(* IEC 61131-3 sources: F100R_S278_Temperville/MyController.device.xml.v3^/Plc Logic.plclogic.xml.v3^/Application.application.xml.v3^/04_PID, 11 files *)

(* ---- A_PincipalRampa.prg.st ---- *)
PROGRAM A_PincipalRampa

IF NOT xTesteResistencias AND NOT xTesteEntradaSaidas THEN
	B_RampaPatamar();
	C_AquecimentoReceita();
ELSE
	E_Termperaturas();
END_IF

(* ---- A_PrincipalPid.prg.st ---- *)
PROGRAM A_PrincipalPid
VAR

END_VAR

IF NOT xTesteResistencias AND NOT xTesteEntradaSaidas THEN
	D_CtrlResistInferiores();
	D_CtrlResistSuperiores();
	//SR_Main();
ELSE
	E_Termperaturas();
END_IF

D_CtrlResist();
C_StandByTemperaturas();
A_TemperaturaGeral();
D_ConvecVentEnt();
D_ConvecVentSai();

(* ---- A_TemperaturaGeral.prg.st ---- *)
PROGRAM A_TemperaturaGeral
VAR
	IndexGTI: INT;
	IndexGPI: INT;
	IndexGTS: INT;
	IndexGPS: INT;
	IndexGTIS: INT;
	IndexGPIS: INT;
	IndexGTSS: INT;
	IndexGPSS: INT;
END_VAR

// ATUALIZAÇÃO DAS TEMPERATURAS E PERCENTAGENS PELA TEMPERATURA GERAL

IF NOT xBloqueioCargaEnvioRec THEN
	// Temperaturas Inferiores
	IF rSetTemperaturaInferiorGeral <> rSetTemperaturaInferiorGeralAux THEN
		FOR IndexGTI:=1 TO iNumResistencias DO
			rSetTemperaturaInferior[IndexGTI]:=rSetTemperaturaInferiorGeral;
		END_FOR
		rSetTemperaturaInferiorGeralAux:=rSetTemperaturaInferiorGeral;
	END_IF

	//Percentagens Inferiores
	IF rSetPorcentagemInferiorGeral <> rSetPorcentagemInferiorGeralAux THEN
		FOR IndexGPI:=1 TO iNumResistencias DO
			rSetPorcentagemInferior[IndexGPI]:=rSetPorcentagemInferiorGeral;
		END_FOR
		rSetPorcentagemInferiorGeralAux:=rSetPorcentagemInferiorGeral;
	END_IF

	//Temperaturas Superiores
	IF rSetTemperaturaSuperiorGeral <> rSetTemperaturaSuperiorGeralAux THEN
		FOR IndexGTS:=1 TO iNumResistencias DO
			rSetTemperaturaSuperior[IndexGTS]:=rSetTemperaturaSuperiorGeral;
		END_FOR
		rSetTemperaturaSuperiorGeralAux:=rSetTemperaturaSuperiorGeral;
	END_IF

	//Percentagens Superiores
	IF rSetPorcentagemSuperiorGeral <> rSetPorcentagemSuperiorGeralAux THEN
		FOR IndexGPS:=1 TO iNumResistencias DO
			rSetPorcentagemSuperior[IndexGPS]:=rSetPorcentagemSuperiorGeral;
		END_FOR
		rSetPorcentagemSuperiorGeralAux:=rSetPorcentagemSuperiorGeral;
	END_IF
END_IF

// INCREMENTA/DECREMENTA MESMO VALOR EM TODAS AS TEMPERATURAS

// Temperaturas Inferiores
	IF xBtHabIncremento THEN
		FOR IndexGTIS:=1 TO iNumResistencias DO
			rSetTemperaturaInferior[IndexGTIS]:=rSetTemperaturaInferior[IndexGTIS]+rIncrementoTemperInf;
			rSetPorcentagemInferior[IndexGTIS]:=rSetPorcentagemInferior[IndexGTIS]+rIncrementoPotenciaInf;
			rSetTemperaturaSuperior[IndexGTIS]:=rSetTemperaturaSuperior[IndexGTIS]+rIncrementoTemperSup;
			rSetPorcentagemSuperior[IndexGTIS]:=rSetPorcentagemSuperior[IndexGTIS]+rIncrementoPotenciaSup;
		END_FOR
		xBtHabIncremento:=FALSE;
	END_IF

	//IF xBtIncrTemperInfSub THEN
	//	FOR IndexGTIS:=1 TO iNumResistencias DO
	//		rSetTemperaturaInferior[IndexGTIS]:=rSetTemperaturaInferior[IndexGTIS]-rIncrementoTemper;
	//	END_FOR
	//	xBtIncrTemperInfSub:=FALSE;
	//END_IF

// Percentagens Inferiores
	//IF xBtIncrPercentInfAdd THEN
	//	FOR IndexGPIS:=1 TO 25 DO
	//		rSetPorcentagemInferior[IndexGPIS]:=rSetPorcentagemInferior[IndexGPIS]+rIncrementoTemper;
	//	END_FOR
	//	xBtIncrPercentInfAdd:=FALSE;
	//END_IF

	//IF xBtIncrPercentInfSub THEN
	//	FOR IndexGPIS:=1 TO 25 DO
	//		rSetPorcentagemInferior[IndexGPIS]:=rSetPorcentagemInferior[IndexGPIS]-rIncrementoTemper;
	//	END_FOR
	//	xBtIncrPercentInfSub:=FALSE;
	//END_IF

// Temperaturas Superiores
	//IF xBtIncrTemperSupAdd THEN
	//	FOR IndexGTSS:=1 TO 25 DO
	//		rSetTemperaturaSuperior[IndexGTSS]:=rSetTemperaturaSuperior[IndexGTSS]+rIncrementoTemper;
	//	END_FOR
	//	xBtIncrTemperSupAdd:=FALSE;
	//END_IF

	//IF xBtIncrTemperSupSub THEN
	//	FOR IndexGTSS:=1 TO 25 DO
	//		rSetTemperaturaSuperior[IndexGTSS]:=rSetTemperaturaSuperior[IndexGTSS]-rIncrementoTemper;
	//	END_FOR
	//	xBtIncrTemperSupSub:=FALSE;
	//END_IF

// Percentagens Superiores
	//IF xBtIncrPercentSupAdd THEN
	//	FOR IndexGPSS:=1 TO 25 DO
	//		rSetPorcentagemSuperior[IndexGPSS]:=rSetPorcentagemSuperior[IndexGPSS]+rIncrementoTemper;
	//	END_FOR
	//	xBtIncrPercentSupAdd:=FALSE;
	//END_IF

	//IF xBtIncrPercentSupSub THEN
	//	FOR IndexGPSS:=1 TO 25 DO
	//		rSetPorcentagemSuperior[IndexGPSS]:=rSetPorcentagemSuperior[IndexGPSS]-rIncrementoTemper;
	//	END_FOR
	//	xBtIncrPercentSupSub:=FALSE;
	//END_IF

(* ---- B_RampaPatamar.prg.st ---- *)
PROGRAM B_RampaPatamar
VAR
	PassoRampaPat: INT;
	xIniciaRampa01: BOOL;
	xIniciaRampa02: BOOL;
	xIniciaRampa03: BOOL;
	xIniciaPatamar01: BOOL;
	xIniciaPatamar02: BOOL;
	xIniciaPatamar03: BOOL;
	xFimRampa01: BOOL;
	xFimRampa02: BOOL;
	xFimRampa03: BOOL;
	xFimPatamar01: BOOL;
	xFimPatamar02: BOOL;
	xFimPatamar03: BOOL;
	xFimRampaAquecimento: BOOL;
	rTempoTotalAquecimento: REAL;
	wStatusRampaAquecimento: WORD;
	rTempoFinalRampa01: REAL;
	rTempoFinalRampa02: REAL;
	rTempoFinalRampa03: REAL;
	rTempoFinalPatamar01: REAL;
	rTempoFinalPatamar02: REAL;
	rTempoFinalPatamar03: REAL;
	wStatusRampa01: WORD;
	wStatusRampa02: WORD;
	wStatusRampa03: WORD;
	wStatusPatamar01: WORD;
	wStatusPatamar02: WORD;
	wStatusPatamar03: WORD;
	///rHisterese01: REAL;
	///rHisterese02: REAL;
	///rHisterese03: REAL;
	/// Parametros de Entrada
	xIniciaAquecimentoRampa: BOOL;
	rTemperaturaPatamar01: REAL;
	rTemperaturaPatamar02: REAL;
	rTemperaturaPatamar03: REAL;
	rTempoPatamar01: REAL;
	rTempoPatamar02: REAL;
	rTempoPatamar03: REAL;
	rTempoTotalAquecimentoProgramado: REAL;
	///////////////////////////////////////////////////////////
	Index: INT;
	IndexR01: INT;
	IndexR02: INT;
	IndexR03: INT;
	IndexP01: INT;
	IndexP02: INT;
	IndexP03: INT;
	IndexT: INT;
	IndexTl: INT;
	TermoparRampa: ARRAY[1..100] OF INT;
	TermoparRampaInf: ARRAY[1..50] OF INT;
	TermoparRampaSup: ARRAY[1..50] OF INT;
	fbRampa01: ARRAY[1..100] OF Rampa;
	///fbRampa02: ARRAY [1..100] OF Rampa;
	///fbRampa03: ARRAY [1..100] OF Rampa;
	fbPatamar01: ARRAY[1..100] OF Patamar;
	///fbPatamar02: ARRAY [1..100] OF Patamar;
	///fbPatamar03: ARRAY [1..100] OF Patamar;
	rTempoRampa01Decor: REAL;
	rTempoRampa02Decor: REAL;
	rTempoRampa03Decor: REAL;
	rTempoPatamar01Decor: REAL;
	rTempoPatamar02Decor: REAL;
	rTempoPatamar03Decor: REAL;
	rTempoRampa01Decorrido: REAL;
	rTempoRampa02Decorrido: REAL;
	rTempoRampa03Decorrido: REAL;
	rTempoPatamar01Decorrido: REAL;
	rTempoPatamar02Decorrido: REAL;
	rTempoPatamar03Decorrido: REAL;
	rTempoAquecimentoDecorrido: REAL;
	TempoRealRampa01: TON;
	TempoRealRampa01In: BOOL;
	TempoRealRampa01Pt: TIME;
	TempoRealRampa01Et: TIME;
	TempoRealRampa01Q: BOOL;
	TempoRealRampa02: TON;
	TempoRealRampa02In: BOOL;
	TempoRealRampa02Pt: TIME;
	TempoRealRampa02Et: TIME;
	TempoRealRampa02Q: BOOL;
	TempoRealRampa03: TON;
	TempoRealRampa03In: BOOL;
	TempoRealRampa03Pt: TIME;
	TempoRealRampa03Et: TIME;
	TempoRealRampa03Q: BOOL;
	TempoRealPatamar01: TON;
	TempoRealPatamar01In: BOOL;
	TempoRealPatamar01Pt: TIME;
	TempoRealPatamar01Et: TIME;
	TempoRealPatamar01Q: BOOL;
	TempoRealPatamar02: TON;
	TempoRealPatamar02In: BOOL;
	TempoRealPatamar02Pt: TIME;
	TempoRealPatamar02Et: TIME;
	TempoRealPatamar02Q: BOOL;
	TempoRealPatamar03: TON;
	TempoRealPatamar03In: BOOL;
	TempoRealPatamar03Pt: TIME;
	TempoRealPatamar03Et: TIME;
	TempoRealPatamar03Q: BOOL;
	xFimRampa001: ARRAY[1..100] OF BOOL;
	///xFimRampa002: ARRAY [1..100] OF BOOL;
	///xFimRampa003: ARRAY [1..100] OF BOOL;
	xFimPatamar001: ARRAY[1..100] OF BOOL;
	///xFimPatamar002: ARRAY [1..100] OF BOOL;
	///xFimPatamar003: ARRAY [1..100] OF BOOL;
	xIniciaRampa001: ARRAY[1..100] OF BOOL;
	///xIniciaRampa002: ARRAY [1..100] OF BOOL;
	///xIniciaRampa003: ARRAY [1..100] OF BOOL;
	xIniciaPatamar001: ARRAY[1..100] OF BOOL;
	///xIniciaPatamar002: ARRAY [1..100] OF BOOL;
	///xIniciaPatamar003: ARRAY [1..100] OF BOOL;
	xSaidaRampa01: ARRAY[1..100] OF BOOL;
	///xSaidaRampa02: ARRAY [1..100] OF BOOL;
	///xSaidaRampa03: ARRAY [1..100] OF BOOL;
	xSaidaPatamar01: ARRAY[1..100] OF BOOL;
	///xSaidaPatamar02: ARRAY [1..100] OF BOOL;
	///xSaidaPatamar03: ARRAY [1..100] OF BOOL;
	xSaidaReleRampPatam: ARRAY[1..100] OF BOOL;
	xFimRampa01Soma: INT;
	xFimRampa02Soma: INT;
	xFimRampa03Soma: INT;
	xFimPatamar01Soma: INT;
	xFimPatamar02Soma: INT;
	xFimPatamar03Soma: INT;
	Trp01: blink;
	xAlternaSetorRampa: BOOL;
	PulsoLigaResistencias: PulsoPositivo;
	xPulsoDataHoraProgOk: BOOL;
	rConsumoInicialAquec_kW: REAL;

	xDesligaRampaForno: BOOL;
	xFornoEmRampa	: BOOL ;
END_VAR

// Seleção do Tipo de Aquecimento Rampa/Patamar ou Receita

IF xBtSelAqueceRampaReceita THEN
	xAqueceRampaPatamar:=TRUE;
	xAqueceReceita:=FALSE;
	xBtSelAqueceRapidoLento:=FALSE;
ELSE
	xAqueceRampaPatamar:=FALSE;
	xAqueceReceita:=TRUE;
END_IF

IF xAqueceRampaPatamar THEN
	uStatusSelAquecimento:=1;
END_IF
IF xAqueceReceita AND xAqueceRapido THEN
	uStatusSelAquecimento:=2;
END_IF
IF xAqueceReceita AND xAqueceLento THEN
	uStatusSelAquecimento:=3;
END_IF

// Ligamento pela Programação Horaria

PulsoLigaResistencias(Entrada:=xDataHoraProgOk , SaidaPulsoPo=>xPulsoDataHoraProgOk );

// Aquecimento por Rampa e Patamar

IF xBtLigaAquecimentoRampa THEN
	rTempoRampa03 := rRampaPrincipal;
	xBtLigaResRampa:=TRUE;
	//xBtLigaAquecimentoRampa:=FALSE;
END_IF

IF xBtLigaAquecimentoRampa OR xPulsoDataHoraProgOk THEN
	xIniciaAquecimentoRampa:=TRUE;
	xBtLigaAquecimentoRampa:=FALSE;
END_IF

IF rTempoRampa03<1800 THEN
	rTempoRampa03:=1800;
ELSE
	rTempoRampa03:=rTempoRampa03;
END_IF

// RAMPA PATAMAR GERAL

CASE PassoRampaPat OF
// Inicio Aquecimento
	0:	IF xIniciaAquecimentoRampa THEN
			IndexR01:= 1;
			PassoRampaPat:=5;
		END_IF
// Rampa 01
	5:	xIniciaAquecimentoRampa:=FALSE;
		xIniciaRelatorioAquecRampa:=TRUE;
		xResistenciasLigadas:=TRUE;
		xFornoEmRampa:=TRUE;
		xCmdIniciaCiclo:=TRUE;
		wStatusRampaAquecimento:=1;
		uStatusAquecimento:=1;// Aquecendo
		wStatusRampa01:=1;
		TempoRealRampa01Pt:=T#24H;
		TempoRealRampa01In:=TRUE;
		xIniciaRampa01:=TRUE;
		FOR IndexR01:= 1 TO iNumeroResistencias DO
			xIniciaRampa001[IndexR01]:=xIniciaRampa01;
		END_FOR
		rConsumoInicialAquec_kW:=rConsumoEnergiaReal_kWh;(*Ativo*)

		PassoRampaPat:=6;

	6:	xIniciaRampa01:=FALSE;
		IF xFimRampa01 THEN (* Fim da Rampa de todos os termopares *)
			PassoRampaPat:=7;
		END_IF

	7:	rTempoFinalRampa01:=rTempoRampa01Decor;
		wStatusRampa01:=2;
		PassoRampaPat:=8;

	8:	TempoRealRampa01In:=FALSE;
		PassoRampaPat:=9;

// Patamar 01
	9:	IndexP01:= 1;
		PassoRampaPat:=10;

	10:	xIniciaPatamar01:=TRUE;
		wStatusPatamar01:=1;
		TempoRealPatamar01Pt:=T#24H;
		TempoRealPatamar01In:=TRUE;
		FOR IndexP01:= 1 TO iNumeroResistencias DO
			xIniciaPatamar001[IndexP01]:=xIniciaPatamar01;
		END_FOR
		PassoRampaPat:=11;

	11:	xIniciaPatamar01:=FALSE;
		IF xFimPatamar01 THEN (* Fim Patamar 01*)
			PassoRampaPat:=12;
		END_IF

	12:	rTempoFinalPatamar01:=rTempoPatamar01Decor;
		wStatusPatamar01:=2;
		PassoRampaPat:=13;

	13:	TempoRealPatamar01In:=FALSE;
		PassoRampaPat:=34;//14;
(*
// Rampa 02
	14:	IndexR02:= 1;
		PassoRampaPat:=15;

	15:	xIniciaRampa02:=TRUE;
		wStatusRampa02:=1;
		TempoRealRampa02Pt:=T#24H;
		TempoRealRampa02In:=TRUE;
		FOR IndexR02:= 1 TO iNumeroResistencias DO
			xIniciaRampa002[IndexR02]:=xIniciaRampa02;
		END_FOR
		PassoRampaPat:=16;

	16: xIniciaRampa02:=FALSE;
		IF xFimRampa02 THEN
			PassoRampaPat:=17;
		END_IF

	17:	rTempoFinalRampa02:=rTempoRampa02Decor;
		wStatusRampa02:=2;
		PassoRampaPat:=18;

	18:	TempoRealRampa02In:=FALSE;
		PassoRampaPat:=19;

// Patamar 02
	19:	IndexP02:= 1;
		PassoRampaPat:=20;

	20:	xIniciaPatamar02:=TRUE;
		wStatusPatamar02:=1;
		TempoRealPatamar02Pt:=T#24H;
		TempoRealPatamar02In:=TRUE;
		FOR IndexP02:= 1 TO iNumeroResistencias DO
			xIniciaPatamar002[IndexP02]:=xIniciaPatamar02;
		END_FOR
		PassoRampaPat:=21;

	21:	xIniciaPatamar02:=FALSE;
		IF xFimPatamar02 THEN
			PassoRampaPat:=22;
		END_IF

	22:	rTempoFinalPatamar02:=rTempoPatamar02Decor;
		wStatusPatamar02:=2;
		PassoRampaPat:=23;

	23:	TempoRealPatamar02In:=FALSE;
		PassoRampaPat:=25;

// Rampa 03
	24:	IndexR03:= 1;
		PassoRampaPat:=25;

	25:	xIniciaRampa03:=TRUE;
		wStatusRampa03:=1;
		TempoRealRampa03Pt:=T#24H;
		TempoRealRampa03In:=TRUE;
		FOR IndexR03:= 1 TO iNumeroResistencias DO
			xIniciaRampa003[IndexR03]:=xIniciaRampa03;
		END_FOR
		PassoRampaPat:=26;

	26:	xIniciaRampa03:=FALSE;
		IF xFimRampa03 THEN
			PassoRampaPat:=27;
		END_IF

	27:	rTempoFinalRampa03:=rTempoRampa03Decor;
		wStatusRampa03:=2;
		PassoRampaPat:=28;

	28:	TempoRealRampa03In:=FALSE;
		PassoRampaPat:=29;

// Patamar 03
	29: IndexP03:= 1;
		PassoRampaPat:=30;

	30:	xIniciaPatamar03:=TRUE;
		wStatusPatamar03:=1;
		TempoRealPatamar03Pt:=T#24H;
		TempoRealPatamar03In:=TRUE;
		FOR IndexP03:= 1 TO iNumeroResistencias DO
			xIniciaPatamar001[IndexP03]:=xIniciaPatamar01;
		END_FOR
		PassoRampaPat:=31;

	31:	xIniciaPatamar03:=FALSE;
		IF xFimPatamar03 THEN
			PassoRampaPat:=32;
		END_IF

	32:	rTempoFinalPatamar03:=rTempoPatamar03Decor;
		wStatusPatamar03:=2;
		PassoRampaPat:=33;

	33:	TempoRealPatamar03In:=FALSE;
		PassoRampaPat:=34;*)

// Fim Aquecimento
	34:	xFornoEmRampa:=FALSE;
		xFinalizaRelatorioAquecRampa:=TRUE;
		PassoRampaPat:=35;

	35:	xFimRampaAquecimento:=TRUE;
		xFimAquecimento:=TRUE;
		LigaInfPorAquecimentoRampa:=FALSE; // inclusão 19/08/2020
		LigaSupPorAquecimentoRampa:=FALSE; // inclusão 19/08/2020
		rTempoTotalAquecimento:=rTempoAquecimentoDecorrido;
		wStatusRampaAquecimento:=2;//QUENTE
		uStatusAquecimento:=2;
		//PassoRampaPat:=0;

END_CASE

//Consumo de Energia por Aquecimento
rConsumoAquecRel:= rConsumoEnergiaReal_kWh-rConsumoInicialAquec_kW;

TempoRealRampa01(IN:=TempoRealRampa01In , PT:=TempoRealRampa01Pt , Q=> TempoRealRampa01Q, ET=>TempoRealRampa01Et );
//TempoRealRampa02(IN:=TempoRealRampa02In , PT:=TempoRealRampa02Pt , Q=> TempoRealRampa02Q, ET=>TempoRealRampa02Et );
//TempoRealRampa03(IN:=TempoRealRampa03In , PT:=TempoRealRampa03Pt , Q=> TempoRealRampa03Q, ET=>TempoRealRampa03Et );
rTempoRampa01Decor:=(TIME_TO_REAL(TempoRealRampa01Et))/1000;
//rTempoRampa02Decor:=(TIME_TO_REAL(TempoRealRampa02Et))/1000;
//rTempoRampa03Decor:=(TIME_TO_REAL(TempoRealRampa03Et))/1000;
rTempoRampa01Decorrido:=rTempoRampa01Decor+(rTempoFinalRampa01);
//rTempoRampa02Decorrido:=rTempoRampa02Decor+(rTempoFinalRampa02);
//rTempoRampa03Decorrido:=rTempoRampa03Decor+(rTempoFinalRampa03);

TempoRealPatamar01(IN:=TempoRealPatamar01In , PT:=TempoRealPatamar01Pt , Q=> TempoRealPatamar01Q, ET=>TempoRealPatamar01Et );
//TempoRealPatamar02(IN:=TempoRealPatamar02In , PT:=TempoRealPatamar02Pt , Q=> TempoRealPatamar02Q, ET=>TempoRealPatamar02Et );
//TempoRealPatamar03(IN:=TempoRealPatamar03In , PT:=TempoRealPatamar03Pt , Q=> TempoRealPatamar03Q, ET=>TempoRealPatamar03Et );
rTempoPatamar01Decor:=(TIME_TO_REAL(TempoRealPatamar01Et))/1000;
//rTempoPatamar02Decor:=(TIME_TO_REAL(TempoRealPatamar02Et))/1000;
//rTempoPatamar03Decor:=(TIME_TO_REAL(TempoRealPatamar03Et))/1000;
rTempoPatamar01Decorrido:=rTempoPatamar01Decor+(rTempoFinalPatamar01);
//rTempoPatamar02Decorrido:=rTempoPatamar02Decor+(rTempoFinalPatamar02);
//rTempoPatamar03Decorrido:=rTempoPatamar03Decor+(rTempoFinalPatamar03);

rTempoAquecimentoDecorrido:=rTempoRampa01Decorrido+rTempoPatamar01Decorrido+rTempoRampa02Decorrido+rTempoPatamar02Decorrido+rTempoRampa03Decorrido+rTempoPatamar03Decorrido;
rTempoTotalAquecimentoProgramado:=rTempoRampa01+rTempoRampa02+rTempoRampa03+rTempoPatamar01+rTempoPatamar02+rTempoPatamar03;

xFimRampa01Soma:=0;
xFimRampa02Soma:=0;
xFimRampa03Soma:=0;
xFimPatamar01Soma:=0;
xFimPatamar02Soma:=0;
xFimPatamar03Soma:=0;

// Artificio para adaptar a Rampa de Aquecimento ao Forno Com diferença no numero de setores Inferior e Superior
TermoparRampaInf[1]:=TermoparLogicoInferior[1];
TermoparRampaInf[2]:=TermoparLogicoInferior[2];
TermoparRampaInf[3]:=TermoparLogicoInferior[3];
TermoparRampaInf[4]:=TermoparLogicoInferior[4];
TermoparRampaInf[5]:=TermoparLogicoInferior[5];
TermoparRampaInf[6]:=TermoparLogicoInferior[6];
TermoparRampaInf[7]:=TermoparLogicoInferior[7];
TermoparRampaInf[8]:=TermoparLogicoInferior[8];
TermoparRampaInf[9]:=TermoparLogicoInferior[9];
TermoparRampaInf[10]:=TermoparLogicoInferior[10];
TermoparRampaInf[11]:=TermoparLogicoInferior[11];
TermoparRampaInf[12]:=TermoparLogicoInferior[12];
TermoparRampaInf[13]:=TermoparLogicoInferior[13];
TermoparRampaInf[14]:=TermoparLogicoInferior[14];
TermoparRampaInf[15]:=TermoparLogicoInferior[15];
TermoparRampaInf[16]:=TermoparLogicoInferior[16];
TermoparRampaInf[17]:=TermoparLogicoInferior[17];
TermoparRampaInf[18]:=TermoparLogicoInferior[18];
TermoparRampaInf[19]:=TermoparLogicoInferior[19];
TermoparRampaInf[20]:=TermoparLogicoInferior[20];
TermoparRampaInf[21]:=TermoparLogicoInferior[21];
TermoparRampaInf[22]:=TermoparLogicoInferior[22];
TermoparRampaInf[23]:=TermoparLogicoInferior[23];
TermoparRampaInf[24]:=TermoparLogicoInferior[24];
TermoparRampaInf[25]:=TermoparLogicoInferior[25];
TermoparRampaInf[26]:=TermoparLogicoInferior[26];
TermoparRampaInf[27]:=TermoparLogicoInferior[27];
TermoparRampaInf[28]:=TermoparLogicoInferior[28];
TermoparRampaInf[29]:=TermoparLogicoInferior[29];
TermoparRampaInf[30]:=TermoparLogicoInferior[30];
TermoparRampaInf[31]:=TermoparLogicoInferior[31];
TermoparRampaInf[32]:=TermoparLogicoInferior[32];
TermoparRampaInf[33]:=TermoparLogicoInferior[33];
TermoparRampaInf[34]:=TermoparLogicoInferior[34];
TermoparRampaInf[35]:=TermoparLogicoInferior[35];
TermoparRampaInf[36]:=TermoparLogicoInferior[36];
TermoparRampaInf[37]:=TermoparLogicoInferior[37];
TermoparRampaInf[38]:=TermoparLogicoInferior[38];
TermoparRampaInf[39]:=TermoparLogicoInferior[39];
TermoparRampaInf[40]:=TermoparLogicoInferior[40];
TermoparRampaInf[41]:=TermoparLogicoInferior[41];
TermoparRampaInf[42]:=TermoparLogicoInferior[42];
TermoparRampaInf[43]:=TermoparLogicoInferior[43];
TermoparRampaInf[44]:=TermoparLogicoInferior[44];
TermoparRampaInf[45]:=TermoparLogicoInferior[45];
TermoparRampaInf[46]:=TermoparLogicoInferior[46];
TermoparRampaInf[47]:=TermoparLogicoInferior[47];
TermoparRampaInf[48]:=TermoparLogicoInferior[48];
TermoparRampaInf[49]:=TermoparLogicoInferior[49];
TermoparRampaInf[50]:=TermoparLogicoInferior[50];

TermoparRampaSup[1]:=TermoparLogicoSuperior[1];
TermoparRampaSup[2]:=TermoparLogicoSuperior[2];
TermoparRampaSup[3]:=TermoparLogicoSuperior[3];
TermoparRampaSup[4]:=TermoparLogicoSuperior[4];
TermoparRampaSup[5]:=TermoparLogicoSuperior[5];
TermoparRampaSup[6]:=TermoparLogicoSuperior[6];
TermoparRampaSup[7]:=TermoparLogicoSuperior[7];
TermoparRampaSup[8]:=TermoparLogicoSuperior[8];
TermoparRampaSup[9]:=TermoparLogicoSuperior[9];
TermoparRampaSup[10]:=TermoparLogicoSuperior[10];
TermoparRampaSup[11]:=TermoparLogicoSuperior[11];
TermoparRampaSup[12]:=TermoparLogicoSuperior[12];
TermoparRampaSup[13]:=TermoparLogicoSuperior[13];
TermoparRampaSup[14]:=TermoparLogicoSuperior[14];
TermoparRampaSup[15]:=TermoparLogicoSuperior[15];
TermoparRampaSup[16]:=TermoparLogicoSuperior[16];
TermoparRampaSup[17]:=TermoparLogicoSuperior[17];
TermoparRampaSup[18]:=TermoparLogicoSuperior[18];
TermoparRampaSup[19]:=TermoparLogicoSuperior[19];
TermoparRampaSup[20]:=TermoparLogicoSuperior[20];
TermoparRampaSup[21]:=TermoparLogicoSuperior[21];
TermoparRampaSup[22]:=TermoparLogicoSuperior[22];
TermoparRampaSup[23]:=TermoparLogicoSuperior[23];
TermoparRampaSup[24]:=TermoparLogicoSuperior[24];
TermoparRampaSup[25]:=TermoparLogicoSuperior[25];
TermoparRampaSup[26]:=TermoparLogicoSuperior[26];
TermoparRampaSup[27]:=TermoparLogicoSuperior[27];
TermoparRampaSup[28]:=TermoparLogicoSuperior[28];
TermoparRampaSup[29]:=TermoparLogicoSuperior[29];
TermoparRampaSup[30]:=TermoparLogicoSuperior[30];
TermoparRampaSup[31]:=TermoparLogicoSuperior[31];
TermoparRampaSup[32]:=TermoparLogicoSuperior[32];
TermoparRampaSup[33]:=TermoparLogicoSuperior[33];
TermoparRampaSup[34]:=TermoparLogicoSuperior[34];
TermoparRampaSup[35]:=TermoparLogicoSuperior[35];
TermoparRampaSup[36]:=TermoparLogicoSuperior[36];
TermoparRampaSup[37]:=TermoparLogicoSuperior[37];
TermoparRampaSup[38]:=TermoparLogicoSuperior[38];
TermoparRampaSup[39]:=TermoparLogicoSuperior[39];
TermoparRampaSup[40]:=TermoparLogicoSuperior[40];
TermoparRampaSup[41]:=TermoparLogicoSuperior[41];
TermoparRampaSup[42]:=TermoparLogicoSuperior[42];
TermoparRampaSup[43]:=TermoparLogicoSuperior[43];
TermoparRampaSup[44]:=TermoparLogicoSuperior[44];
TermoparRampaSup[45]:=TermoparLogicoSuperior[45];
TermoparRampaSup[46]:=TermoparLogicoSuperior[46];
TermoparRampaSup[47]:=TermoparLogicoSuperior[47];
TermoparRampaSup[48]:=TermoparLogicoSuperior[48];
TermoparRampaSup[49]:=TermoparLogicoSuperior[49];
TermoparRampaSup[50]:=TermoparLogicoSuperior[50];

//--------------------------------------------------------------------------------------------------------------
FOR IndexT:= 1 TO iNumResistencias DO
	TermoparRampa[IndexT]:=TermoparRampaInf[IndexT];
	TermoparRampa[IndexT+iNumResistencias]:=TermoparRampaSup[IndexT];
END_FOR

FOR Index:= 1 TO iNumeroResistencias DO

// Rampa 01

	xIniciaRampa001[Index]:=xIniciaRampa01;

fbRampa01[Index](
	rTemopar:= 		(INT_TO_REAL(TermoparRampa[Index]))/10,
	rTempMedia:=	rMediaLogicaTemperaturaTotal,
	rPatamar:= 		rSetTemperaturaRampa,//0,
	rTempoRampa:= 	rTempoRampa03,//1,
	xDesabilitaZn:= NOT xResistenciaHabilitada[Index],
	xFimTotRampa:= 	xFimRampa01,
	xIniciaRampa:= 	xIniciaRampa001[Index],
	xFimRampa:= 	xFimRampa001[Index],
	xResetBloco:= 	xDesligaRampaForno,
	xSaida=> 		xSaidaRampa01[Index] );

xFimRampa01Soma:= xFimRampa01Soma+ BOOL_TO_INT (xFimRampa001[Index]);

// Patamar 01
	xIniciaPatamar001[Index]:=xIniciaPatamar01;

fbPatamar01[Index](
	rTemopar:= 		(INT_TO_REAL(TermoparRampa[Index]))/10,
	rPatamar:= 		rSetTemperaturaRampa,//0,
	rHisterese:= 	0.1,
	rTempoPatamar:= 1,
	xDesabilitaZn:= NOT xResistenciaHabilitada[Index],
	xIniciaPatamar:= xIniciaPatamar001[Index],
	xFimPatamar:= 	xFimPatamar001[Index],
	xResetBloco:= 	xDesligaRampaForno,
	xSaida=> 		xSaidaPatamar01[Index]);

xFimPatamar01Soma:= xFimPatamar01Soma+ BOOL_TO_INT (xFimPatamar001[Index]);
(*
// Rampa 02
	xIniciaRampa002[Index]:=xIniciaRampa02;

fbRampa02[Index](
	rTemopar:= 		(INT_TO_REAL(TermoparRampa[Index]))/10,
	rTempMedia:=	rMediaLogicaTemperaturaTotal,
	rPatamar:= 		0,
	rTempoRampa:= 	1,
	xDesabilitaZn:= NOT xResistenciaHabilitada[Index],
	xFimTotRampa:=  xFimRampa02,
	xIniciaRampa:= 	xIniciaRampa002[Index],
	xFimRampa:= 	xFimRampa002[Index],
	xResetBloco:= 	xBtDesligaAquecimento,
	xSaida=> 		xSaidaRampa02[Index] );

xFimRampa02Soma:= xFimRampa02Soma+ BOOL_TO_INT (xFimRampa002[Index]);

// Patamar 02

	xIniciaPatamar002[Index]:=xIniciaPatamar02;

fbPatamar02[Index](
	rTemopar:= 		(INT_TO_REAL(TermoparRampa[Index]))/10,
	rPatamar:= 		0,
	rHisterese:= 	0.1,
	rTempoPatamar:= 1,
	xDesabilitaZn:= NOT xResistenciaHabilitada[Index],
	xIniciaPatamar:= xIniciaPatamar002[Index],
	xFimPatamar:= 	xFimPatamar002[Index],
	xResetBloco:= 	xBtDesligaAquecimento,
	xSaida=> 		xSaidaPatamar02[Index]);

xFimPatamar02Soma:= xFimPatamar02Soma+ BOOL_TO_INT (xFimPatamar002[Index]);

// Rampa 03
	xIniciaRampa003[Index]:=xIniciaRampa03;

fbRampa03[Index](
	rTemopar:= 		(INT_TO_REAL(TermoparRampa[Index]))/10,
	rTempMedia:=	rMediaLogicaTemperaturaTotal,
	rPatamar:= 		rSetTemperaturaInferiorGeral,
	rTempoRampa:= 	rTempoRampa03,
	xDesabilitaZn:= NOT xResistenciaHabilitada[Index],
	xFimTotRampa:=  xFimRampa03,
	xIniciaRampa:= 	xIniciaRampa003[Index],
	xFimRampa:= 	xFimRampa003[Index],
	xResetBloco:= 	xBtDesligaAquecimento,
	xSaida=> 		xSaidaRampa03[Index] );

xFimRampa03Soma:= xFimRampa03Soma+ BOOL_TO_INT (xFimRampa003[Index]);

// Patamar 03

	xIniciaPatamar003[Index]:=xIniciaPatamar03;

fbPatamar03[Index](
	rTemopar:= 		(INT_TO_REAL(TermoparRampa[Index]))/10,
	rPatamar:= 		rSetTemperaturaInferiorGeral,
	rHisterese:= 	0.1,
	rTempoPatamar:= 1,//rTempoPatamar03,
	xDesabilitaZn:= NOT xResistenciaHabilitada[Index],
	xIniciaPatamar:= xIniciaPatamar003[Index],
	xFimPatamar:= 	xFimPatamar003[Index],
	xResetBloco:= 	xBtDesligaAquecimento,
	xSaida=> 		xSaidaPatamar03[Index]);

xFimPatamar03Soma:= xFimPatamar03Soma+ BOOL_TO_INT (xFimPatamar003[Index]);
*)
xSaidaReleRampPatam[Index]:=xSaidaRampa01[Index] (*OR xSaidaRampa02[Index] OR xSaidaRampa03[Index]*) OR xSaidaPatamar01[Index] (*OR xSaidaPatamar02[Index] OR xSaidaPatamar03[Index]*);

END_FOR

xFimRampa01:= xFimRampa01Soma=iNumeroResistencias;
//xFimRampa02:= xFimRampa02Soma=iNumeroResistencias;
//xFimRampa03:= xFimRampa03Soma=iNumeroResistencias;
xFimPatamar01:= xFimPatamar01Soma=iNumeroResistencias;
//xFimPatamar02:= xFimPatamar02Soma=iNumeroResistencias;
//xFimPatamar03:= xFimPatamar03Soma=iNumeroResistencias;

//Fim da Rampa de Aquecimento

xDesligaRampaForno:=xBtDesligaAquecimento  OR xSemEnergia OR xOperacaoManual OR xTempoDesligaResistQ OR xBtEmergencia;
IF xDesligaRampaForno AND xFornoEmRampa THEN
	xFinalizaRelatorioAquecRampa:=TRUE;
END_IF

IF xDesligaRampaForno THEN
	    xIniciaAquecimentoRampa:=FALSE;
		xFimRampaAquecimento:=FALSE;
		xIniciaRampa01:=FALSE;
		TempoRealRampa01In:=FALSE;
		TempoRealRampa02In:=FALSE;
		TempoRealRampa03In:=FALSE;
		TempoRealPatamar01In:=FALSE;
		TempoRealPatamar02In:=FALSE;
		TempoRealPatamar03In:=FALSE;
		rTempoTotalAquecimento:=0;
		rTempoFinalRampa01:=0;
		rTempoFinalRampa02:=0;
		rTempoFinalRampa03:=0;
		rTempoFinalPatamar01:=0;
		rTempoFinalPatamar02:=0;
		rTempoFinalPatamar03:=0;
		wStatusRampaAquecimento:=0;
		wStatusRampa01:=0;
		wStatusRampa02:=0;
		wStatusRampa03:=0;
		wStatusPatamar01:=0;
		wStatusPatamar02:=0;
		wStatusPatamar03:=0;
		PassoRampaPat:=0;
		xFornoEmRampa:=FALSE;
		xBtLigaAquecimento:=FALSE;
END_IF

LigaInfPorAquecimentoRampa:=xFimRampaAquecimento;
LigaSupPorAquecimentoRampa:=xFimRampaAquecimento;

// Tempo de Alternancia entre Zonas
Trp01(ENABLE:= TRUE, TIMELOW:= T#1S, TIMEHIGH:= T#1S, OUT=> xAlternaSetorRampa );

xSaidaReleRampaPatamarInf[1]:= xSaidaReleRampPatam[1] AND xResistenciaHabilitadaInferior[1] AND xAlternaSetorRampa;
xSaidaReleRampaPatamarInf[2]:= xSaidaReleRampPatam[2] AND xResistenciaHabilitadaInferior[2] AND NOT xAlternaSetorRampa;
xSaidaReleRampaPatamarInf[3]:= xSaidaReleRampPatam[3] AND xResistenciaHabilitadaInferior[3] AND xAlternaSetorRampa;
xSaidaReleRampaPatamarInf[4]:= xSaidaReleRampPatam[4] AND xResistenciaHabilitadaInferior[4] AND NOT xAlternaSetorRampa;
xSaidaReleRampaPatamarInf[5]:= xSaidaReleRampPatam[5] AND xResistenciaHabilitadaInferior[5] AND  xAlternaSetorRampa;
xSaidaReleRampaPatamarInf[6]:= xSaidaReleRampPatam[6] AND xResistenciaHabilitadaInferior[6] AND NOT xAlternaSetorRampa;
xSaidaReleRampaPatamarInf[7]:= xSaidaReleRampPatam[7] AND xResistenciaHabilitadaInferior[7] AND  xAlternaSetorRampa;
xSaidaReleRampaPatamarInf[8]:= xSaidaReleRampPatam[8] AND xResistenciaHabilitadaInferior[8] AND NOT xAlternaSetorRampa;
xSaidaReleRampaPatamarInf[9]:= xSaidaReleRampPatam[9] AND xResistenciaHabilitadaInferior[9] AND xAlternaSetorRampa;
xSaidaReleRampaPatamarInf[10]:= xSaidaReleRampPatam[10] AND xResistenciaHabilitadaInferior[10] AND NOT xAlternaSetorRampa;
xSaidaReleRampaPatamarInf[11]:= xSaidaReleRampPatam[11] AND xResistenciaHabilitadaInferior[11] AND NOT xAlternaSetorRampa;
xSaidaReleRampaPatamarInf[12]:= xSaidaReleRampPatam[12] AND xResistenciaHabilitadaInferior[12] AND  xAlternaSetorRampa;
xSaidaReleRampaPatamarInf[13]:= xSaidaReleRampPatam[13] AND xResistenciaHabilitadaInferior[13] AND NOT xAlternaSetorRampa;
xSaidaReleRampaPatamarInf[14]:= xSaidaReleRampPatam[14] AND xResistenciaHabilitadaInferior[14] AND xAlternaSetorRampa;
xSaidaReleRampaPatamarInf[15]:= xSaidaReleRampPatam[15] AND xResistenciaHabilitadaInferior[15] AND NOT xAlternaSetorRampa;
xSaidaReleRampaPatamarInf[16]:= xSaidaReleRampPatam[16] AND xResistenciaHabilitadaInferior[16] AND xAlternaSetorRampa;
xSaidaReleRampaPatamarInf[17]:= xSaidaReleRampPatam[17] AND xResistenciaHabilitadaInferior[17] AND NOT xAlternaSetorRampa;
xSaidaReleRampaPatamarInf[18]:= xSaidaReleRampPatam[18] AND xResistenciaHabilitadaInferior[18] AND xAlternaSetorRampa;
xSaidaReleRampaPatamarInf[19]:= xSaidaReleRampPatam[19] AND xResistenciaHabilitadaInferior[19] AND NOT xAlternaSetorRampa;
xSaidaReleRampaPatamarInf[20]:= xSaidaReleRampPatam[20] AND xResistenciaHabilitadaInferior[20] AND  xAlternaSetorRampa;
xSaidaReleRampaPatamarInf[21]:= xSaidaReleRampPatam[21] AND xResistenciaHabilitadaInferior[21] AND  xAlternaSetorRampa;
xSaidaReleRampaPatamarInf[22]:= xSaidaReleRampPatam[22] AND xResistenciaHabilitadaInferior[22] AND NOT xAlternaSetorRampa;
xSaidaReleRampaPatamarInf[23]:= xSaidaReleRampPatam[23] AND xResistenciaHabilitadaInferior[23] AND  xAlternaSetorRampa;
xSaidaReleRampaPatamarInf[24]:= xSaidaReleRampPatam[24] AND xResistenciaHabilitadaInferior[24] AND NOT xAlternaSetorRampa;
xSaidaReleRampaPatamarInf[25]:= xSaidaReleRampPatam[25] AND xResistenciaHabilitadaInferior[25] AND  xAlternaSetorRampa;
xSaidaReleRampaPatamarInf[26]:= xSaidaReleRampPatam[26] AND xResistenciaHabilitadaInferior[26] AND NOT xAlternaSetorRampa;
xSaidaReleRampaPatamarInf[27]:= xSaidaReleRampPatam[27] AND xResistenciaHabilitadaInferior[27] AND  xAlternaSetorRampa;
xSaidaReleRampaPatamarInf[28]:= xSaidaReleRampPatam[28] AND xResistenciaHabilitadaInferior[28] AND NOT xAlternaSetorRampa;
xSaidaReleRampaPatamarInf[29]:= xSaidaReleRampPatam[29] AND xResistenciaHabilitadaInferior[29] AND  xAlternaSetorRampa;
xSaidaReleRampaPatamarInf[30]:= xSaidaReleRampPatam[30] AND xResistenciaHabilitadaInferior[30] AND NOT xAlternaSetorRampa;
xSaidaReleRampaPatamarInf[31]:= xSaidaReleRampPatam[31] AND xResistenciaHabilitadaInferior[31] AND NOT xAlternaSetorRampa;
xSaidaReleRampaPatamarInf[32]:= xSaidaReleRampPatam[32] AND xResistenciaHabilitadaInferior[32] AND  xAlternaSetorRampa;
xSaidaReleRampaPatamarInf[33]:= xSaidaReleRampPatam[33] AND xResistenciaHabilitadaInferior[33] AND NOT xAlternaSetorRampa;
xSaidaReleRampaPatamarInf[34]:= xSaidaReleRampPatam[34] AND xResistenciaHabilitadaInferior[34] AND  xAlternaSetorRampa;
xSaidaReleRampaPatamarInf[35]:= xSaidaReleRampPatam[35] AND xResistenciaHabilitadaInferior[35] AND NOT xAlternaSetorRampa;
xSaidaReleRampaPatamarInf[36]:= xSaidaReleRampPatam[36] AND xResistenciaHabilitadaInferior[36] AND  xAlternaSetorRampa;
xSaidaReleRampaPatamarInf[37]:= xSaidaReleRampPatam[37] AND xResistenciaHabilitadaInferior[37] AND NOT xAlternaSetorRampa;
xSaidaReleRampaPatamarInf[38]:= xSaidaReleRampPatam[38] AND xResistenciaHabilitadaInferior[38] AND  xAlternaSetorRampa;
xSaidaReleRampaPatamarInf[39]:= xSaidaReleRampPatam[39] AND xResistenciaHabilitadaInferior[39] AND NOT xAlternaSetorRampa;
xSaidaReleRampaPatamarInf[40]:= xSaidaReleRampPatam[40] AND xResistenciaHabilitadaInferior[40] AND  xAlternaSetorRampa;
xSaidaReleRampaPatamarInf[41]:= xSaidaReleRampPatam[41] AND xResistenciaHabilitadaInferior[41] AND  xAlternaSetorRampa;
xSaidaReleRampaPatamarInf[42]:= xSaidaReleRampPatam[42] AND xResistenciaHabilitadaInferior[42] AND NOT xAlternaSetorRampa;
xSaidaReleRampaPatamarInf[43]:= xSaidaReleRampPatam[43] AND xResistenciaHabilitadaInferior[43] AND  xAlternaSetorRampa;
xSaidaReleRampaPatamarInf[44]:= xSaidaReleRampPatam[44] AND xResistenciaHabilitadaInferior[44] AND NOT xAlternaSetorRampa;
xSaidaReleRampaPatamarInf[45]:= xSaidaReleRampPatam[45] AND xResistenciaHabilitadaInferior[45] AND  xAlternaSetorRampa;
xSaidaReleRampaPatamarInf[46]:= xSaidaReleRampPatam[46] AND xResistenciaHabilitadaInferior[46] AND NOT xAlternaSetorRampa;
xSaidaReleRampaPatamarInf[47]:= xSaidaReleRampPatam[47] AND xResistenciaHabilitadaInferior[47] AND  xAlternaSetorRampa;
xSaidaReleRampaPatamarInf[48]:= xSaidaReleRampPatam[48] AND xResistenciaHabilitadaInferior[48] AND NOT xAlternaSetorRampa;
xSaidaReleRampaPatamarInf[49]:= xSaidaReleRampPatam[49] AND xResistenciaHabilitadaInferior[49] AND  xAlternaSetorRampa;
xSaidaReleRampaPatamarInf[50]:= xSaidaReleRampPatam[50] AND xResistenciaHabilitadaInferior[50] AND NOT xAlternaSetorRampa;

xSaidaReleRampaPatamarSup[1]:= xSaidaReleRampPatam[1+iNumResistencias] AND xResistenciaHabilitadaSuperior[1] AND NOT xAlternaSetorRampa;
xSaidaReleRampaPatamarSup[2]:= xSaidaReleRampPatam[2+iNumResistencias] AND xResistenciaHabilitadaSuperior[2] AND xAlternaSetorRampa;
xSaidaReleRampaPatamarSup[3]:= xSaidaReleRampPatam[3+iNumResistencias] AND xResistenciaHabilitadaSuperior[3] AND NOT xAlternaSetorRampa;
xSaidaReleRampaPatamarSup[4]:= xSaidaReleRampPatam[4+iNumResistencias] AND xResistenciaHabilitadaSuperior[4] AND xAlternaSetorRampa;
xSaidaReleRampaPatamarSup[5]:= xSaidaReleRampPatam[5+iNumResistencias] AND xResistenciaHabilitadaSuperior[5] AND NOT xAlternaSetorRampa;
xSaidaReleRampaPatamarSup[6]:= xSaidaReleRampPatam[6+iNumResistencias] AND xResistenciaHabilitadaSuperior[6] AND  xAlternaSetorRampa;
xSaidaReleRampaPatamarSup[7]:= xSaidaReleRampPatam[7+iNumResistencias] AND xResistenciaHabilitadaSuperior[7] AND NOT xAlternaSetorRampa;
xSaidaReleRampaPatamarSup[8]:= xSaidaReleRampPatam[8+iNumResistencias] AND xResistenciaHabilitadaSuperior[8] AND  xAlternaSetorRampa;
xSaidaReleRampaPatamarSup[9]:= xSaidaReleRampPatam[9+iNumResistencias] AND xResistenciaHabilitadaSuperior[9] AND NOT xAlternaSetorRampa;
xSaidaReleRampaPatamarSup[10]:= xSaidaReleRampPatam[10+iNumResistencias] AND xResistenciaHabilitadaSuperior[10] AND xAlternaSetorRampa;
xSaidaReleRampaPatamarSup[11]:= xSaidaReleRampPatam[11+iNumResistencias] AND xResistenciaHabilitadaSuperior[11] AND xALternaSetorRampa;
xSaidaReleRampaPatamarSup[12]:= xSaidaReleRampPatam[12+iNumResistencias] AND xResistenciaHabilitadaSuperior[12] AND NOT xAlternaSetorRampa;
xSaidaReleRampaPatamarSup[13]:= xSaidaReleRampPatam[13+iNumResistencias] AND xResistenciaHabilitadaSuperior[13] AND xAlternaSetorRampa;
xSaidaReleRampaPatamarSup[14]:= xSaidaReleRampPatam[14+iNumResistencias] AND xResistenciaHabilitadaSuperior[14] AND NOT xAlternaSetorRampa;
xSaidaReleRampaPatamarSup[15]:= xSaidaReleRampPatam[15+iNumResistencias] AND xResistenciaHabilitadaSuperior[15] AND xAlternaSetorRampa;
xSaidaReleRampaPatamarSup[16]:= xSaidaReleRampPatam[16+iNumResistencias] AND xResistenciaHabilitadaSuperior[16] AND NOT xAlternaSetorRampa;
xSaidaReleRampaPatamarSup[17]:= xSaidaReleRampPatam[17+iNumResistencias] AND xResistenciaHabilitadaSuperior[17] AND xAlternaSetorRampa;
xSaidaReleRampaPatamarSup[18]:= xSaidaReleRampPatam[18+iNumResistencias] AND xResistenciaHabilitadaSuperior[18] AND NOT xAlternaSetorRampa;
xSaidaReleRampaPatamarSup[19]:= xSaidaReleRampPatam[19+iNumResistencias] AND xResistenciaHabilitadaSuperior[19] AND xAlternaSetorRampa;
xSaidaReleRampaPatamarSup[20]:= xSaidaReleRampPatam[20+iNumResistencias] AND xResistenciaHabilitadaSuperior[20] AND NOT xAlternaSetorRampa;
xSaidaReleRampaPatamarSup[21]:= xSaidaReleRampPatam[21+iNumResistencias] AND xResistenciaHabilitadaSuperior[21] AND NOT xAlternaSetorRampa;
xSaidaReleRampaPatamarSup[22]:= xSaidaReleRampPatam[22+iNumResistencias] AND xResistenciaHabilitadaSuperior[22] AND xAlternaSetorRampa;
xSaidaReleRampaPatamarSup[23]:= xSaidaReleRampPatam[23+iNumResistencias] AND xResistenciaHabilitadaSuperior[23] AND NOT xAlternaSetorRampa;
xSaidaReleRampaPatamarSup[24]:= xSaidaReleRampPatam[24+iNumResistencias] AND xResistenciaHabilitadaSuperior[24] AND xAlternaSetorRampa;
xSaidaReleRampaPatamarSup[25]:= xSaidaReleRampPatam[25+iNumResistencias] AND xResistenciaHabilitadaSuperior[25] AND NOT xAlternaSetorRampa;
xSaidaReleRampaPatamarSup[26]:= xSaidaReleRampPatam[26+iNumResistencias] AND xResistenciaHabilitadaSuperior[26] AND xAlternaSetorRampa;
xSaidaReleRampaPatamarSup[27]:= xSaidaReleRampPatam[27+iNumResistencias] AND xResistenciaHabilitadaSuperior[27] AND NOT xAlternaSetorRampa;
xSaidaReleRampaPatamarSup[28]:= xSaidaReleRampPatam[28+iNumResistencias] AND xResistenciaHabilitadaSuperior[28] AND xAlternaSetorRampa;
xSaidaReleRampaPatamarSup[29]:= xSaidaReleRampPatam[29+iNumResistencias] AND xResistenciaHabilitadaSuperior[29] AND NOT xAlternaSetorRampa;
xSaidaReleRampaPatamarSup[30]:= xSaidaReleRampPatam[30+iNumResistencias] AND xResistenciaHabilitadaSuperior[30] AND xAlternaSetorRampa;
xSaidaReleRampaPatamarSup[31]:= xSaidaReleRampPatam[31+iNumResistencias] AND xResistenciaHabilitadaSuperior[31] AND xAlternaSetorRampa;
xSaidaReleRampaPatamarSup[32]:= xSaidaReleRampPatam[32+iNumResistencias] AND xResistenciaHabilitadaSuperior[32] AND NOT xAlternaSetorRampa;
xSaidaReleRampaPatamarSup[33]:= xSaidaReleRampPatam[33+iNumResistencias] AND xResistenciaHabilitadaSuperior[33] AND xAlternaSetorRampa;
xSaidaReleRampaPatamarSup[34]:= xSaidaReleRampPatam[34+iNumResistencias] AND xResistenciaHabilitadaSuperior[34] AND NOT xAlternaSetorRampa;
xSaidaReleRampaPatamarSup[35]:= xSaidaReleRampPatam[35+iNumResistencias] AND xResistenciaHabilitadaSuperior[35] AND xAlternaSetorRampa;
xSaidaReleRampaPatamarSup[36]:= xSaidaReleRampPatam[36+iNumResistencias] AND xResistenciaHabilitadaSuperior[36] AND NOT xAlternaSetorRampa;
xSaidaReleRampaPatamarSup[37]:= xSaidaReleRampPatam[37+iNumResistencias] AND xResistenciaHabilitadaSuperior[37] AND  xAlternaSetorRampa;
xSaidaReleRampaPatamarSup[38]:= xSaidaReleRampPatam[38+iNumResistencias] AND xResistenciaHabilitadaSuperior[38] AND NOT xAlternaSetorRampa;
xSaidaReleRampaPatamarSup[39]:= xSaidaReleRampPatam[39+iNumResistencias] AND xResistenciaHabilitadaSuperior[39] AND  xAlternaSetorRampa;
xSaidaReleRampaPatamarSup[40]:= xSaidaReleRampPatam[40+iNumResistencias] AND xResistenciaHabilitadaSuperior[40] AND NOT xAlternaSetorRampa;
xSaidaReleRampaPatamarSup[41]:= xSaidaReleRampPatam[41+iNumResistencias] AND xResistenciaHabilitadaSuperior[41] AND NOT xAlternaSetorRampa;
xSaidaReleRampaPatamarSup[42]:= xSaidaReleRampPatam[42+iNumResistencias] AND xResistenciaHabilitadaSuperior[42] AND xAlternaSetorRampa;
xSaidaReleRampaPatamarSup[43]:= xSaidaReleRampPatam[43+iNumResistencias] AND xResistenciaHabilitadaSuperior[43] AND NOT xAlternaSetorRampa;
xSaidaReleRampaPatamarSup[44]:= xSaidaReleRampPatam[44+iNumResistencias] AND xResistenciaHabilitadaSuperior[44] AND xAlternaSetorRampa;
xSaidaReleRampaPatamarSup[45]:= xSaidaReleRampPatam[45+iNumResistencias] AND xResistenciaHabilitadaSuperior[45] AND NOT xAlternaSetorRampa;
xSaidaReleRampaPatamarSup[46]:= xSaidaReleRampPatam[46+iNumResistencias] AND xResistenciaHabilitadaSuperior[46] AND xAlternaSetorRampa;
xSaidaReleRampaPatamarSup[47]:= xSaidaReleRampPatam[47+iNumResistencias] AND xResistenciaHabilitadaSuperior[47] AND NOT xAlternaSetorRampa;
xSaidaReleRampaPatamarSup[48]:= xSaidaReleRampPatam[48+iNumResistencias] AND xResistenciaHabilitadaSuperior[48] AND xAlternaSetorRampa;
xSaidaReleRampaPatamarSup[49]:= xSaidaReleRampPatam[49+iNumResistencias] AND xResistenciaHabilitadaSuperior[49] AND NOT xAlternaSetorRampa;
xSaidaReleRampaPatamarSup[50]:= xSaidaReleRampPatam[50+iNumResistencias] AND xResistenciaHabilitadaSuperior[50] AND xAlternaSetorRampa;

(* ------------------ ESCRITA DA RECEITA ----------------------------*)

IF iHabilitaEscritaReceitaAquec=1 THEN
	iEscreverReceitaAquecim:=1;
	iHabilitaEscritaReceitaAquec:=0;
END_IF

IF iEscreverReceitaAquecim=1 THEN

	iReceitaAquecimEscritaOk:=1;
	iEscreverReceitaAquecim:=0;

	xReceitaAqiecimCarregadaOk:=TRUE;

END_IF

(* ---- C_AquecimentoReceita.prg.st ---- *)
PROGRAM C_AquecimentoReceita
VAR
	Index: INT;
	PulsoLigaResistSupLento: PulsoPositivo;
	PulsoLigaResistSupRapid: PulsoPositivo;
	xTempoDesligaResist: TON;
	TemperaturaSetPointInferior: ARRAY[1..60] OF AlarmeTemperatura;
	TemperaturaSetPointSuperior: ARRAY[1..60] OF AlarmeTemperatura;
	xTemperaturaSetorInferiorOk: ARRAY[1..60] OF BOOL;
	xTemperaturaSetorSuperiorOk: ARRAY[1..60] OF BOOL;
	iSomaSetorInferiorOk: INT;
	iSomaSetorSuperiorOk: INT;
	xSetorInferiorQuente: BOOL;
	xSetorSuperiorQuente: BOOL;
	xFimAquecimentoReceita: BOOL;
	xPulsoLigaResistSupLento: BOOL;
	xPulsoLigaResistSupRapid: BOOL;
	xTempoDesligaResistIn: BOOL;
END_VAR

// Aquecimento por Rampa e Patamar

IF (xBtLigaAquecimento)(* OR xDataHoraProgOk) AND xAqueceReceita*) THEN
	xBtLigaResCiclo:=TRUE;
	xIniciaAquecimentoRec:=TRUE;
	//xCmdIniciaCiclo:=TRUE;
END_IF

IF	xBtLigaAquecimento (*AND xAqueceReceita*) THEN
	xBtLigaAquecimento:=FALSE;
END_IF

IF xIniciaAquecimentoRec THEN
	xAuxiliarLigaResistenciasInferiores:=TRUE;
	xResistenciasLigadas:=TRUE;
	xCmdIniciaCiclo:=TRUE;
	xIniciaRelatorioAquecRec:=TRUE;
	uStatusAquecimento:=1;
	xIniciaAquecimentoRec:=FALSE;
END_IF

iSomaSetorInferiorOk:=0;
iSomaSetorSuperiorOk:=0;
FOR Index:= 1 TO iNumResistencias DO
// Temperatura Inferior
	TemperaturaSetPointInferior[Index](
		TermoparAtual:= 			TermoparLogicoInferior[Index]/10,
		TemperaturaMax:= 			rSetTemperaturaInferior[Index],
		ResetAlarm:= 				xBtDesligaAquecimento OR NOT xResistenciasLigadas,
		TermoparAlmTemperatura=> 	xTemperaturaSetorInferiorOk[Index]);

	iSomaSetorInferiorOk:=iSomaSetorInferiorOk + BOOL_TO_INT(xTemperaturaSetorInferiorOk[Index]);

// Temperatura Superior
	TemperaturaSetPointSuperior[Index](
		TermoparAtual:= 			TermoparLogicoSuperior[Index]/10,
		TemperaturaMax:= 			rSetTemperaturaSuperior[Index],
		ResetAlarm:= 				xBtDesligaAquecimento OR NOT xResistenciasLigadas,
		TermoparAlmTemperatura=> 	xTemperaturaSetorSuperiorOk[Index]);

	iSomaSetorSuperiorOk:=iSomaSetorSuperiorOk + BOOL_TO_INT(xTemperaturaSetorSuperiorOk[Index]);

	xSetorInferiorQuente:=iSomaSetorInferiorOk=iNumResistencias;
	xSetorSuperiorQuente:=iSomaSetorSuperiorOk=iNumResistencias;

END_FOR

xFimAquecimentoReceita:=xSetorInferiorQuente AND xSetorSuperiorQuente;

IF xFimAquecimentoReceita (*and xAqueceReceita*) THEN
	uStatusAquecimento:=2;
	xFimAquecimento:=TRUE;
	xFinalizaRelatorioAquecRec:=TRUE;
END_IF

//Pulso Liga Resistências Superiores

PulsoLigaResistSupLento(Entrada:= xSetorInferiorQuente, 				SaidaPulsoPo=> xPulsoLigaResistSupLento);
PulsoLigaResistSupRapid(Entrada:= xAuxiliarLigaResistenciasInferiores , SaidaPulsoPo=> xPulsoLigaResistSupRapid);

// Seleção do Aquecimento por Receita Rapido ou Lento

xAqueceLento:= FALSE;//NOT xBtSelAqueceRapidoLento AND xAqueceReceita;
xAqueceRapido:= TRUE;//xBtSelAqueceRapidoLento AND xAqueceReceita;

// Aquecimento Rápido
IF xAqueceRapido AND xPulsoLigaResistSupRapid THEN
	xAuxiliarLigaResistenciasSuperiores:=TRUE;
END_IF
// Aquecimento Lento
IF xAqueceLento AND xPulsoLigaResistSupLento THEN
	xAuxiliarLigaResistenciasSuperiores:=TRUE;
END_IF

// Desliga Resistência se Motor do forno não Rodando

IF NOT xMotorFornoLigado AND NOT xFornoEmCicloComCarga AND xResistenciasLigadas THEN
	xTempoDesligaResistIn:=TRUE;
ELSE
	xTempoDesligaResistIn:=FALSE;
END_IF

xTempoDesligaResist(IN:=xTempoDesligaResistIn , PT:=T#10S , Q=>xTempoDesligaResistQ , ET=> );

// Desligamento das Resistências
IF xBtDesligaAquecimento OR xSemEnergia OR xOperacaoManual OR xTempoDesligaResistQ OR xBtEmergencia THEN
	xAuxiliarLigaResistenciasInferiores:=FALSE;
	xAuxiliarLigaResistenciasSuperiores:=FALSE;
	xResistenciasLigadas:=FALSE;
	xIniciaAquecimentoRec:=FALSE;
	uStatusAquecimento:=0;
	xFimAquecimento:=FALSE;
	xCmFinalizaCiclo:=TRUE;
	//xDesligaAquecimento:=FALSE;
END_IF
IF xBtDesligaAquecimento (*AND xAqueceReceita*) THEN
	xBtDeslResCiclo:=true;
	xBtDesligaAquecimento:=FALSE;
END_IF

LigaInfPorAquecimentoReceita:= xAuxiliarLigaResistenciasInferiores;
LigaSupPorAquecimentoReceita:= xAuxiliarLigaResistenciasSuperiores;

(* ---- C_StandByTemperaturas.prg.st ---- *)
PROGRAM C_StandByTemperaturas
VAR
	Index: INT;
	IndexGTI: INT;
	IndexGPI: INT;
	IndexGTS: INT;
	IndexGPS: INT;
	rSpInferiorStandby: REAL;
	rSpSuperiorStandby: REAL;
	xSetTempStandyByCiclo: BOOL;
	xTonSetTemperStdBy: BOOL;
	TonSetTemperStdBy: TON;
	xTonSetTemperStdByIn: BOOL;
	xTonSetTemperStdByQ: BOOL;
	tTonSetTemperStdByPt: TIME;
	tTonSetTemperStdByEt: TIME;
	xAbortaStandByCiclo: BOOL;
	rSetTemperaturaInferiorGeralAux: REAL;
	rSetTemperaturaSuperiorGeralAux: REAL;
	rSetPorcentagemInferiorGeralAux: REAL;
	rSetPorcentagemSuperiorGeralAux: REAL;
END_VAR

//xAbortaStandByCiclo:=BtAbortaStandByCiclo;

IF BtAbortaStandByCiclo THEN
	xAbortaStandByCiclo:=TRUE;
END_IF

IF 	xFimDescForIniStdBy OR xSetTempStandyByInicio THEN
	xTonSetTemperStdBy:=TRUE;
	xFimDescForIniStdBy:=FALSE;
	xSetTempStandyByInicio:=FALSE;
	xAbortaStandByCiclo:=FALSE;//
END_IF

IF 	xTonSetTemperStdBy AND NOT xAbortaStandByCiclo and not xStdByTemperaturaDesabilit THEN
	xTonSetTemperStdByIn := TRUE;
ELSE
	xTonSetTemperStdByIn := FALSE;
END_IF;

tTonSetTemperStdByPt:=DINT_TO_TIME (INT_TO_DINT(iTempoIniStdByTemperatura)*1000);

TonSetTemperStdBy(IN:= xTonSetTemperStdByIn, PT:=tTonSetTemperStdByPt , Q=> xTonSetTemperStdByQ, ET=>tTonSetTemperStdByEt );

iTempoStdByTemperDecorrido:=DINT_TO_INT(TIME_TO_DINT (tTonSetTemperStdByEt)/1000);

IF iTempoIniStdByTemperatura<>0 THEN
	xStdByTemperaturaHabilitado:=TRUE;
ELSE
	xStdByTemperaturaHabilitado:=FALSE;
END_IF

xStdByTemperaturaDesabilit:= NOT xStdByTemperaturaHabilitado;

xSetTempStandyByCiclo:=xTonSetTemperStdByQ;
xImgSetTempStandByCiclo:=xSetTempStandyByCiclo;

IF xStartCargaForno OR xOperacaoManual OR xFornoEmEspera THEN
	xTonSetTemperStdBy:=FALSE;
	xStartCargaForno:=FALSE;
END_IF

IF BtAbortaStandByCiclo THEN
	BtAbortaStandByCiclo:=FALSE;
END_IF

rSpInferiorStandby:=rSetPointInferiorStandby;
rSpSuperiorStandby:=rSetPointSuperiorStandby;

FOR Index:=1 TO iNumResistencias DO
	IF xSetTempStandyByCiclo THEN
		rSetPointTemperaturaInferior[Index]:=rSpInferiorStandby;
		rSetPointTemperaturaSuperior[Index]:=rSpSuperiorStandby;
	ELSE
		rSetPointTemperaturaInferior[Index]:=rSetTemperaturaInferior[Index];
		rSetPointTemperaturaSuperior[Index]:=rSetTemperaturaSuperior[Index];
	END_IF;
END_FOR

(* ---- D_ConvecVentEnt.prg.st ---- *)
PROGRAM D_ConvecVentEnt
VAR
	PassoVentConvecEnt: INT;
	PassoPauseVentConvecEnt: INT;
	PassoAlmVentConvecEnt: INT;
	PassoManualVentConvecEnt: INT;
	///Blocos Nativos
	///Blocos Criados
	ControleSsrConveccaoEnt: PidPwm;
	HabResConveccaoEnt: HabilitaDesabilita;
	ReleDefeitoConvecEntSsr01: AlarmeRelesSsr;
	ReleDefeitoConvecEntSsr02: AlarmeRelesSsr;
	ReleDefeitoConvecEntSsr03: AlarmeRelesSsr;
	xExecutaVentConvecEnt: BOOL;
	xExecutaStopVentConvecEnt: BOOL;
	xStopVentConvecEntDone: BOOL;
	iVelocidadeVentConvecEnt: INT;
	rTermoparVentConvecEntLeitura: REAL;
	rTermoparVentConvecEntControle: REAL;
	rSetPointTemperaturaConveccaoEnt: REAL;
	xLigaDesligaResistConvecEnt: BOOL;
	xLigaDesligaVentConvecEnt: BOOL;

	xLigaMotorConveccaoEnt: BOOL;

	xAlarmeSsr01ConvecEntSon: BOOL;
	xAlarmeSsr02ConvecEntSon: BOOL;
	xAlarmeSsr03ConvecEntSon: BOOL;

END_VAR

// CONVEÇÃO FONÇADA COM VENTILADOR

//Lógica Ventilador

CASE PassoVentConvecEnt OF

		0:	PassoVentConvecEnt:=2;

		2: 	IF xLigaDesligaResistConvecEnt THEN
				PassoVentConvecEnt:=10;
			END_IF
			IF rTemperaturaConveccaoEnt>=150 THEN
				PassoVentConvecEnt:=50;
			END_IF

		10: iVelocidadeVentConvecEnt:=iVelocidadeStbVentConvecEnt;
			PassoVentConvecEnt:=15;

		15:	xLigaMotorConveccaoEnt:=TRUE;
			PassoVentConvecEnt:=20;

		20: PassoVentConvecEnt:=25;

		21: IF (rTemperaturaConveccaoEnt>150) THEN
				PassoVentConvecEnt:=50;
			END_IF
			IF iVelocidadeVentConvecEnt<>iVelocidadeStbVentConvecEnt THEN
				PassoVentConvecEnt:=10;
			END_IF
			IF NOT xLigaDesligaResistConvecEnt THEN
				PassoVentConvecEnt:=25;
			END_IF
			IF xPause THEN
				PassoPauseVentConvecEnt:=10;
				PassoVentConvecEnt:=300;
			END_IF
			IF xAlarmeMotorVentConvecEnt THEN
				PassoAlmVentConvecEnt:=10;
				PassoVentConvecEnt:=400;
			END_IF

		25: IF (rTemperaturaConveccaoEnt<130) THEN
				PassoVentConvecEnt:=30;
			END_IF
			IF xLigaDesligaResistConvecEnt THEN
				PassoVentConvecEnt:=50;
			END_IF
			IF xPause THEN
				PassoPauseVentConvecEnt:=10;
				PassoVentConvecEnt:=300;
			END_IF
			IF xAlarmeMotorVentConvecEnt THEN
				PassoAlmVentConvecEnt:=10;
				PassoVentConvecEnt:=400;
			END_IF

		30: xLigaMotorConveccaoEnt:=FALSE;
			PassoVentConvecEnt:=35;

		35: PassoVentConvecEnt:=0;

		50:	iVelocidadeVentConvecEnt:=iVelocidadeJogVentConvecEnt;
			PassoVentConvecEnt:=55;

		55: xLigaMotorConveccaoEnt:=TRUE;
			PassoVentConvecEnt:=60;

		60: PassoVentConvecEnt:=65;

		65: IF iVelocidadeVentConvecEnt<>iVelocidadeJogVentConvecEnt THEN
				PassoVentConvecEnt:=50;
			END_IF
			IF NOT xLigaDesligaResistConvecEnt THEN
				PassoVentConvecEnt:=70;
			END_IF
			IF xPause THEN
				PassoPauseVentConvecEnt:=50;
				PassoVentConvecEnt:=300;
			END_IF
			IF xAlarmeMotorVentConvecEnt THEN
				PassoAlmVentConvecEnt:=50;
				PassoVentConvecEnt:=400;
			END_IF

		70: iVelocidadeVentConvecEnt:=iVelocidadeStbVentConvecEnt;
			PassoVentConvecEnt:=75;

		75:	PassoVentConvecEnt:=80;

		80: PassoVentConvecEnt:=25;

		// Emergência Pausa/Reinicio
		300:xLigaMotorConveccaoEnt:=FALSE;
			PassoVentConvecEnt:=301;

		301:PassoVentConvecEnt:=302;

		302:IF xRestart THEN
				PassoVentConvecEnt:=303;
			END_IF

		303:PassoVentConvecEnt:=PassoPauseVentConvecEnt;

		// Alarme Motor Parada/Reinicio
		400:xLigaMotorConveccaoEnt:=FALSE;
			PassoVentConvecEnt:=401;

		401:PassoVentConvecEnt:=402;

		402:IF xRestart AND iCanOpenInverConvecEntStateOk THEN
				PassoVentConvecEnt:=PassoAlmVentConvecEnt;
			END_IF

END_CASE

// MOVIMENTAÇÃO PELO COMANDO ENTRADAS DIGITAIS DO INVERSOR
// Comando e Direção
xMotorConveccaoEnt:=xLigaMotorConveccaoEnt;

InversorConvecEnt.i_xAvanco:=xMotorConveccaoEnt;

// Velocidade
InversorConvecEnt.i_iFreqRef:=iVelocidadeVentConvecEnt;
//------------------------------------------------------------------------\\

IF xOperacaoManual THEN
	PassoVentConvecEnt:=0;
	PassoPauseVentConvecEnt:=0;
	PassoAlmVentConvecEnt:=0;
	PassoManualVentConvecEnt:=0;
	xExecutaVentConvecEnt:=FALSE;
	xLigaMotorConveccaoEnt:=FALSE;
END_IF

// CONTROLE DE TEMPERATURA
rTermoparVentConvecEntLeitura:=INT_TO_REAL(TermoparConveccaoEnt)/10;
rTermoparVentConvecEntControle:=INT_TO_REAL(TermoparConveccaoEnt)/10;
rSetPointTemperaturaConveccaoEnt:=INT_TO_REAL(iSetPointTemperaturaConveccaoEnt);

//HabResConveccaoEnt(
//			Alarme01:= 	(*xAlarmeResistRompidaInferior[Index]*),
//			Alarme02:= 	,//AlmTermoparAbertoLogicoInf[Index],
//			Alarme03:=	,//AlmTemperaturaExcedeuLogicoInf[Index],
//			Entrada:= 	BtHabDesabResistConveccaoEnt,
//			Entrada02:=	,//BtHabilitaResistenciasGeralInferior OR TpHabilitaResistenciasOnQ,
//			Entrada03:= ,//BtDesabilitaResistenciasGeralInferior OR xDesabilitaSobreTemperInferior OR xDesabilitaSobreTemperSuperior,
//			StatusSaida=> xHabDesabResistConveccaoEnt);

IF BtHabDesabResistConveccaoEnt AND NOT xHabDesabResistConveccaoEnt THEN
	xHabDesabResistConveccaoEnt:=TRUE;
END_IF
IF (BtHabDesabResistConveccaoEnt AND xHabDesabResistConveccaoEnt) OR xAlmTemperExcedeuConvecEntSin OR xAlmTermoparAbertoConvecEntSin THEN
	xHabDesabResistConveccaoEnt:=FALSE;
END_IF

IF (xResistenciasLigadas AND rMediaLogicaTemperaturaTotal>400 AND xHabDesabResistConveccaoEnt) OR xForceLigConvecEntVent THEN
	xLigaDesligaResistConvecEnt:=TRUE;
ELSE
	xLigaDesligaResistConvecEnt:=FALSE;
END_IF

// Setor - Convecção
	ControleSsrConveccaoEnt(
	xLigaDesliga		:=  xLigaDesligaResistConvecEnt AND xMotorVentConvecEntLigado,
	xHabilitaControle	:=  TRUE,//xHabilitaBlocoResistConvec,
	xForceResistencia	:=  FALSE,
	xHabilitaResistencia:=  TRUE,
	AlarmeResistencia	:=	,
	xRstTemperaturaOk	:=	,
	xFornoComCarga		:=	,
	rTermoparLeitura	:= 	rTermoparVentConvecEntLeitura,
	rTermoparControle	:=  rTermoparVentConvecEntControle,
	rSetTemperatura		:= 	rSetPointTemperaturaConveccaoEnt,
	rProcentagem		:= 	100,
	rGanhoPorporcionaKp	:= 	10,//Proporciona
	rGanhoIntegralKi	:= 	50,//Integal
	rGanhoDerivativoKd	:= 	0,//Derivativo
	rTempoCiclo			:=	101,
	xresetPidBlk		:= xResetPid,
	SaidaPwm			=>	xReleSsrConveccaoEnt,
	xTemperaturaOk		=>	,
	rTemperatura		=>	rTemperaturaConveccaoEnt);

xRetornoSsrConveccaoEnt:= xRetornoSsr01ConveccaoEnt OR xRetornoSsr02ConveccaoEnt OR xRetornoSsr03ConveccaoEnt;

ReleDefeitoConvecEntSsr01(
	RetornoReleSsr:= 	xRetornoSsr01ConveccaoEnt,
	ResistRompida:= 	,
	ReleSsr:= 			xReleSsrConveccaoEnt,
	ResetAlarm:= 		bResetAlmGeral,
	AlarmeSsrAberto=> 	xAlarmeSsr01ConvecEntAberto,
	AlarmeSsrFechado=>	xAlarmeSsr01ConvecEntFechado,
	AlarmeSonoro=> 		xAlarmeSsr01ConvecEntSon);

ReleDefeitoConvecEntSsr02(
	RetornoReleSsr:= 	xRetornoSsr02ConveccaoEnt,
	ResistRompida:= 	,
	ReleSsr:= 			xReleSsrConveccaoEnt,
	ResetAlarm:= 		bResetAlmGeral,
	AlarmeSsrAberto=> 	xAlarmeSsr02ConvecEntAberto,
	AlarmeSsrFechado=>	xAlarmeSsr02ConvecEntFechado,
	AlarmeSonoro=> 		xAlarmeSsr02ConvecEntSon);

ReleDefeitoConvecEntSsr03(
	RetornoReleSsr:= 	xRetornoSsr03ConveccaoEnt,
	ResistRompida:= 	,
	ReleSsr:= 			xReleSsrConveccaoEnt,
	ResetAlarm:= 		bResetAlmGeral,
	AlarmeSsrAberto=> 	xAlarmeSsr03ConvecEntAberto,
	AlarmeSsrFechado=>	xAlarmeSsr03ConvecEntFechado,
	AlarmeSonoro=> 		xAlarmeSsr03ConvecEntSon);

xAlarmeSsrConvecEntAberto:= xAlarmeSsr01ConvecEntAberto OR xAlarmeSsr02ConvecEntAberto OR xAlarmeSsr03ConvecEntAberto;
xAlarmeSsrConvecEntFechado:= xAlarmeSsr01ConvecEntFechado OR xAlarmeSsr02ConvecEntFechado OR xAlarmeSsr03ConvecEntFechado;

xAlarmeSsrConvecEntSin:=xAlarmeSsrConvecEntAberto OR xAlarmeSsrConvecEntFechado;
xAlarmeSsrConvecEntSon:=xAlarmeSsr01ConvecEntSon OR xAlarmeSsr02ConvecEntSon OR xAlarmeSsr03ConvecEntSon;

//resistencia 01
	IF NOT xRetornoSsr01ConveccaoEnt THEN
			iAnimaResistenciaSsr01ConvecEnt:=1;(*Resistência Desligada*)
	END_IF
	IF xRetornoSsr01ConveccaoEnt THEN
			iAnimaResistenciaSsr01ConvecEnt:=2; (*Resistência Ligada*)
	END_IF
	IF xAlarmeSsr01ConvecEntAberto THEN
			iAnimaResistenciaSsr01ConvecEnt:=3; (*Resistência Alarme Aberto*)
	END_IF
	IF  xAlarmeSsr01ConvecEntFechado THEN
			iAnimaResistenciaSsr01ConvecEnt:=4; (*Resistência Alarme rele em curto*)
	END_IF
	IF TermoparConvecEntAberto THEN
			iAnimaResistenciaSsr01ConvecEnt:=5; (*Termopar Alarme*)
	END_IF

//resistencia 02
	IF NOT xRetornoSsr02ConveccaoEnt THEN
			iAnimaResistenciaSsr02ConvecEnt:=1;(*Resistência Desligada*)
	END_IF
	IF xRetornoSsr02ConveccaoEnt THEN
			iAnimaResistenciaSsr02ConvecEnt:=2; (*Resistência Ligada*)
	END_IF
	IF xAlarmeSsr02ConvecEntAberto THEN
			iAnimaResistenciaSsr02ConvecEnt:=3; (*Resistência Alarme Aberto*)
	END_IF
	IF  xAlarmeSsr02ConvecEntFechado THEN
			iAnimaResistenciaSsr02ConvecEnt:=4; (*Resistência Alarme rele em curto*)
	END_IF
	IF TermoparConvecEntAberto THEN
			iAnimaResistenciaSsr02ConvecEnt:=5; (*Termopar Alarme*)
	END_IF
//resistencia 03
	IF NOT xRetornoSsr03ConveccaoEnt THEN
			iAnimaResistenciaSsr03ConvecEnt:=1;(*Resistência Desligada*)
	END_IF
	IF xRetornoSsr03ConveccaoEnt THEN
			iAnimaResistenciaSsr03ConvecEnt:=2; (*Resistência Ligada*)
	END_IF
	IF xAlarmeSsr03ConvecEntAberto THEN
			iAnimaResistenciaSsr03ConvecEnt:=3; (*Resistência Alarme Aberto*)
	END_IF
	IF  xAlarmeSsr03ConvecEntFechado THEN
			iAnimaResistenciaSsr03ConvecEnt:=4; (*Resistência Alarme rele em curto*)
	END_IF
	IF TermoparConvecEntAberto THEN
			iAnimaResistenciaSsr03ConvecEnt:=5; (*Termopar Alarme*)
	END_IF

(* ---- D_ConvecVentSai.prg.st ---- *)
PROGRAM D_ConvecVentSai
VAR
	PassoVentConvecSai: INT;
	PassoPauseVentConvecSai: INT;
	PassoAlmVentConvecSai: INT;
	PassoManualVentConvecSai: INT;
	///Blocos Nativos
	///Blocos Criados
	ControleSsrConveccaoSai: PidPwm;
	HabResConveccaoSai: HabilitaDesabilita;
	ReleDefeitoConvecSaiSsr01: AlarmeRelesSsr;
	ReleDefeitoConvecSaiSsr02: AlarmeRelesSsr;
	ReleDefeitoConvecSaiSsr03: AlarmeRelesSsr;
	xExecutaVentConvecSai: BOOL;
	xExecutaStopVentConvecSai: BOOL;
	xStopVentConvecSaiDone: BOOL;
	iVelocidadeVentConvecSai: INT;
	rTermoparVentConvecSaiLeitura: REAL;
	rTermoparVentConvecSaiControle: REAL;
	rSetPointTemperaturaConveccaoSai: REAL;
	xLigaDesligaResistConvecSai: BOOL;
	xLigaDesligaVentConvecSai: BOOL;

	xLigaMotorConveccaoSai: BOOL;

	xAlarmeSsr01ConvecSaiSon: BOOL;
	xAlarmeSsr02ConvecSaiSon: BOOL;
	xAlarmeSsr03ConvecSaiSon: BOOL;

END_VAR

// CONVEÇÃO FONÇADA COM VENTILADOR

//Lógica Ventilador

CASE PassoVentConvecSai OF

		0:	PassoVentConvecSai:=2;

		2: 	IF xLigaDesligaResistConvecSai THEN
				PassoVentConvecSai:=10;
			END_IF
			IF rTemperaturaConveccaoSai>=150 THEN
				PassoVentConvecSai:=50;
			END_IF

		10: iVelocidadeVentConvecSai:=iVelocidadeStbVentConvecSai;
			PassoVentConvecSai:=15;

		15:	xLigaMotorConveccaoSai:=TRUE;
			PassoVentConvecSai:=20;

		20: PassoVentConvecSai:=25;

		21: IF (rTemperaturaConveccaoSai>150) THEN
				PassoVentConvecSai:=50;
			END_IF
			IF iVelocidadeVentConvecSai<>iVelocidadeStbVentConvecSai THEN
				PassoVentConvecSai:=10;
			END_IF
			IF NOT xLigaDesligaResistConvecSai THEN
				PassoVentConvecSai:=25;
			END_IF
			IF xPause THEN
				PassoPauseVentConvecSai:=10;
				PassoVentConvecSai:=300;
			END_IF
			IF xAlarmeMotorVentConvecSai THEN
				PassoAlmVentConvecSai:=10;
				PassoVentConvecSai:=400;
			END_IF

		25: IF (rTemperaturaConveccaoSai<130) THEN
				PassoVentConvecSai:=30;
			END_IF
			IF xLigaDesligaResistConvecSai THEN
				PassoVentConvecSai:=50;
			END_IF
			IF xPause THEN
				PassoPauseVentConvecSai:=10;
				PassoVentConvecSai:=300;
			END_IF
			IF xAlarmeMotorVentConvecSai THEN
				PassoAlmVentConvecSai:=10;
				PassoVentConvecSai:=400;
			END_IF

		30: xLigaMotorConveccaoSai:=FALSE;
			PassoVentConvecSai:=35;

		35: PassoVentConvecSai:=0;

		50:	iVelocidadeVentConvecSai:=iVelocidadeJogVentConvecSai;
			PassoVentConvecSai:=55;

		55: xLigaMotorConveccaoSai:=TRUE;
			PassoVentConvecSai:=60;

		60: PassoVentConvecSai:=65;

		65: IF iVelocidadeVentConvecSai<>iVelocidadeJogVentConvecSai THEN
				PassoVentConvecSai:=50;
			END_IF
			IF NOT xLigaDesligaResistConvecSai THEN
				PassoVentConvecSai:=70;
			END_IF
			IF xPause THEN
				PassoPauseVentConvecSai:=50;
				PassoVentConvecSai:=300;
			END_IF
			IF xAlarmeMotorVentConvecSai THEN
				PassoAlmVentConvecSai:=50;
				PassoVentConvecSai:=400;
			END_IF

		70: iVelocidadeVentConvecSai:=iVelocidadeStbVentConvecSai;
			PassoVentConvecSai:=75;

		75:	PassoVentConvecSai:=80;

		80: PassoVentConvecSai:=25;

		// Emergência Pausa/Reinicio
		300:xLigaMotorConveccaoSai:=FALSE;
			PassoVentConvecSai:=301;

		301:PassoVentConvecSai:=302;

		302:IF xRestart THEN
				PassoVentConvecSai:=303;
			END_IF

		303:PassoVentConvecSai:=PassoPauseVentConvecSai;

		// Alarme Motor Parada/Reinicio
		400:xLigaMotorConveccaoSai:=FALSE;
			PassoVentConvecSai:=401;

		401:PassoVentConvecSai:=402;

		402:IF xRestart AND iCanOpenInverConvecSaiStateOk THEN
				PassoVentConvecSai:=PassoAlmVentConvecSai;
			END_IF

END_CASE

// MOVIMENTAÇÃO PELO COMANDO ENTRADAS DIGITAIS DO INVERSOR
// Comando e Direção
xMotorConveccaoSai:=xLigaMotorConveccaoSai;

InversorConvecSai.i_xAvanco:=xMotorConveccaoSai;

// Velocidade
InversorConvecSai.i_iFreqRef:=iVelocidadeVentConvecSai;
//------------------------------------------------------------------------\\

IF xOperacaoManual THEN
	PassoVentConvecSai:=0;
	PassoPauseVentConvecSai:=0;
	PassoAlmVentConvecSai:=0;
	PassoManualVentConvecSai:=0;
	xExecutaVentConvecSai:=FALSE;
	xLigaMotorConveccaoSai:=FALSE;
END_IF

// CONTROLE DE TEMPERATURA
rTermoparVentConvecSaiLeitura:=INT_TO_REAL(TermoparConveccaoSai)/10;
rTermoparVentConvecSaiControle:=INT_TO_REAL(TermoparConveccaoSai)/10;
rSetPointTemperaturaConveccaoSai:=INT_TO_REAL(iSetPointTemperaturaConveccaoSai);

//HabResConveccaoSai(
//			Alarme01:= 	(*xAlarmeResistRompidaInferior[Index]*),
//			Alarme02:= 	,//AlmTermoparAbertoLogicoInf[Index],
//			Alarme03:=	,//AlmTemperaturaExcedeuLogicoInf[Index],
//			Entrada:= 	BtHabDesabResistConveccaoSai,
//			Entrada02:=	,//BtHabilitaResistenciasGeralInferior OR TpHabilitaResistenciasOnQ,
//			Entrada03:= ,//BtDesabilitaResistenciasGeralInferior OR xDesabilitaSobreTemperInferior OR xDesabilitaSobreTemperSuperior,
//			StatusSaida=> xHabDesabResistConveccaoSai);

IF BtHabDesabResistConveccaoSai AND NOT xHabDesabResistConveccaoSai THEN
	xHabDesabResistConveccaoSai:=TRUE;
END_IF
IF (BtHabDesabResistConveccaoSai AND xHabDesabResistConveccaoSai) OR xAlmTemperExcedeuConvecSaiSin OR xAlmTermoparAbertoConvecSaiSin THEN
	xHabDesabResistConveccaoSai:=FALSE;
END_IF

IF (xResistenciasLigadas AND rMediaLogicaTemperaturaTotal>400 AND xHabDesabResistConveccaoSai) OR xForceLigConvecSaiVent THEN
	xLigaDesligaResistConvecSai:=TRUE;
ELSE
	xLigaDesligaResistConvecSai:=FALSE;
END_IF

// Setor - Convecção
	ControleSsrConveccaoSai(
	xLigaDesliga		:=  xLigaDesligaResistConvecSai AND xMotorVentConvecSaiLigado,
	xHabilitaControle	:=  TRUE,//xHabilitaBlocoResistConvec,
	xForceResistencia	:=  FALSE,
	xHabilitaResistencia:=  TRUE,
	AlarmeResistencia	:=	,
	xRstTemperaturaOk	:=	,
	xFornoComCarga		:=	,
	rTermoparLeitura	:= 	rTermoparVentConvecSaiLeitura,
	rTermoparControle	:=  rTermoparVentConvecSaiControle,
	rSetTemperatura		:= 	rSetPointTemperaturaConveccaoSai,
	rProcentagem		:= 	100,
	rGanhoPorporcionaKp	:= 	10,//Proporciona
	rGanhoIntegralKi	:= 	50,//Integal
	rGanhoDerivativoKd	:= 	0,//Derivativo
	rTempoCiclo			:=	101,
	xresetPidBlk		:= xResetPid,
	SaidaPwm			=>	xReleSsrConveccaoSai,
	xTemperaturaOk		=>	,
	rTemperatura		=>	rTemperaturaConveccaoSai);

xRetornoSsrConveccaoSai:= xRetornoSsr01ConveccaoSai OR xRetornoSsr02ConveccaoSai OR xRetornoSsr03ConveccaoSai;

ReleDefeitoConvecSaiSsr01(
	RetornoReleSsr:= 	xRetornoSsr01ConveccaoSai,
	ResistRompida:= 	,
	ReleSsr:= 			xReleSsrConveccaoSai,
	ResetAlarm:= 		bResetAlmGeral,
	AlarmeSsrAberto=> 	xAlarmeSsr01ConvecSaiAberto,
	AlarmeSsrFechado=>	xAlarmeSsr01ConvecSaiFechado,
	AlarmeSonoro=> 		xAlarmeSsr01ConvecSaiSon);

ReleDefeitoConvecSaiSsr02(
	RetornoReleSsr:= 	xRetornoSsr02ConveccaoSai,
	ResistRompida:= 	,
	ReleSsr:= 			xReleSsrConveccaoSai,
	ResetAlarm:= 		bResetAlmGeral,
	AlarmeSsrAberto=> 	xAlarmeSsr02ConvecSaiAberto,
	AlarmeSsrFechado=>	xAlarmeSsr02ConvecSaiFechado,
	AlarmeSonoro=> 		xAlarmeSsr02ConvecSaiSon);

ReleDefeitoConvecSaiSsr03(
	RetornoReleSsr:= 	xRetornoSsr03ConveccaoSai,
	ResistRompida:= 	,
	ReleSsr:= 			xReleSsrConveccaoSai,
	ResetAlarm:= 		bResetAlmGeral,
	AlarmeSsrAberto=> 	xAlarmeSsr03ConvecSaiAberto,
	AlarmeSsrFechado=>	xAlarmeSsr03ConvecSaiFechado,
	AlarmeSonoro=> 		xAlarmeSsr03ConvecSaiSon);

xAlarmeSsrConvecSaiAberto:= xAlarmeSsr01ConvecSaiAberto OR xAlarmeSsr02ConvecSaiAberto OR xAlarmeSsr03ConvecSaiAberto;
xAlarmeSsrConvecSaiFechado:= xAlarmeSsr01ConvecSaiFechado OR xAlarmeSsr02ConvecSaiFechado OR xAlarmeSsr03ConvecSaiFechado;

xAlarmeSsrConvecSaiSin:=xAlarmeSsrConvecSaiAberto OR xAlarmeSsrConvecSaiFechado;
xAlarmeSsrConvecSaiSon:=xAlarmeSsr01ConvecSaiSon OR xAlarmeSsr02ConvecSaiSon OR xAlarmeSsr03ConvecSaiSon;

//resistencia 01
	IF NOT xRetornoSsr01ConveccaoSai THEN
			iAnimaResistenciaSsr01ConvecSai:=1;(*Resistência Desligada*)
	END_IF
	IF xRetornoSsr01ConveccaoSai THEN
			iAnimaResistenciaSsr01ConvecSai:=2; (*Resistência Ligada*)
	END_IF
	IF xAlarmeSsr01ConvecSaiAberto THEN
			iAnimaResistenciaSsr01ConvecSai:=3; (*Resistência Alarme Aberto*)
	END_IF
	IF  xAlarmeSsr01ConvecSaiFechado THEN
			iAnimaResistenciaSsr01ConvecSai:=4; (*Resistência Alarme rele em curto*)
	END_IF
	IF TermoparConvecSaiAberto THEN
			iAnimaResistenciaSsr01ConvecSai:=5; (*Termopar Alarme*)
	END_IF

//resistencia 02
	IF NOT xRetornoSsr02ConveccaoSai THEN
			iAnimaResistenciaSsr02ConvecSai:=1;(*Resistência Desligada*)
	END_IF
	IF xRetornoSsr02ConveccaoSai THEN
			iAnimaResistenciaSsr02ConvecSai:=2; (*Resistência Ligada*)
	END_IF
	IF xAlarmeSsr02ConvecSaiAberto THEN
			iAnimaResistenciaSsr02ConvecSai:=3; (*Resistência Alarme Aberto*)
	END_IF
	IF  xAlarmeSsr02ConvecSaiFechado THEN
			iAnimaResistenciaSsr02ConvecSai:=4; (*Resistência Alarme rele em curto*)
	END_IF
	IF TermoparConvecSaiAberto THEN
			iAnimaResistenciaSsr02ConvecSai:=5; (*Termopar Alarme*)
	END_IF
//resistencia 03
	IF NOT xRetornoSsr03ConveccaoSai THEN
			iAnimaResistenciaSsr03ConvecSai:=1;(*Resistência Desligada*)
	END_IF
	IF xRetornoSsr03ConveccaoSai THEN
			iAnimaResistenciaSsr03ConvecSai:=2; (*Resistência Ligada*)
	END_IF
	IF xAlarmeSsr03ConvecSaiAberto THEN
			iAnimaResistenciaSsr03ConvecSai:=3; (*Resistência Alarme Aberto*)
	END_IF
	IF  xAlarmeSsr03ConvecSaiFechado THEN
			iAnimaResistenciaSsr03ConvecSai:=4; (*Resistência Alarme rele em curto*)
	END_IF
	IF TermoparConvecSaiAberto THEN
			iAnimaResistenciaSsr03ConvecSai:=5; (*Termopar Alarme*)
	END_IF

(* ---- D_CtrlResist.prg.st ---- *)
PROGRAM D_CtrlResist
VAR
END_VAR

// Tempo de Alternancia entre Zonas
TB01(ENABLE:= TRUE, TIMELOW:= T#2S, TIMEHIGH:= T#2S, OUT=> xAlternaSetor );

// Tempo de Pausa de Resistências
IF xIniciaPausaResistencias THEN
	xIniciaPausaResistInf:=TRUE;
	xIniciaPausaResistSup:=TRUE;
	xIniciaTempoPausaResistSup:=TRUE;
	xIniciaPausaResistencias:=FALSE;
END_IF
// Inferiores
TemporizaPausaResistInferior(
	IniciaTempo:= 	xIniciaPausaResistInf,
	AbortaTempo:= 	,
	SetPointTempo:= iTempoPausaResistInf,
	FimTempo:= 		xFimTempoPausaResistInf,
	TempoDecorrido=> iTempoPausaResistInfDecorrido,
	TempoRestante=> );

IF xIniciaPausaResistInf THEN
	xResistenciaInferiorPausa:=TRUE;
	xIniciaPausaResistInf:=FALSE;
END_IF

IF xFimTempoPausaResistInf THEN
	xResistenciaInferiorPausa:=FALSE;
END_IF

// Superiores
TemporizaPausaResistSuperior(
	IniciaTempo:= 	xIniciaPausaResistSup,
	AbortaTempo:= 	,
	SetPointTempo:= iTempoPausaResistSup,
	FimTempo:= 		xFimTempoPausaResistSup,
	TempoDecorrido=> iTempoPausaResistSupDecorrido,
	TempoRestante=> );

IF xIniciaPausaResistSup THEN
	xResistenciaSuperiorPausa01:=TRUE;
	xIniciaPausaResistSup:=FALSE;
END_IF

IF xFimTempoPausaResistSup THEN
	xResistenciaSuperiorPausa01:=FALSE;
END_IF

//Tempo P/ inicio da Pausa nas Resistências Superiores após a carga

TempoInicioPausa02ResistSuperior(IN:= xIniciaTempoPausaResistSup, PT:= T#1000S, Q=> , ET=> );

iTempoParaInicioPausaDecor:= DINT_TO_INT((TIME_TO_DINT(TempoInicioPausa02ResistSuperior.ET))/1000);

IF  iTempoParaInicioPausaDecor >= iTempoInicioPausa02ResistSup AND NOT xFornoEmEspera THEN
	xIniciaTempoPausaResistSup:=FALSE;
	xIniciaPausa02ResistSup:=TRUE;
END_IF

TemporizaPausa02ResistSuperior(
	IniciaTempo:= 	xIniciaPausa02ResistSup,
	AbortaTempo:= 	,
	SetPointTempo:= iTempoPausa02ResistSup,
	FimTempo:= 		xFimTempoPausa02ResistSup,
	TempoDecorrido=> iTempoPausa02ResistSupDecorrido,
	TempoRestante=> );

IF xIniciaPausa02ResistSup THEN
	xResistenciaSuperiorPausa02:=TRUE;
	xIniciaPausa02ResistSup:=FALSE;
END_IF

IF xFimTempoPausa02ResistSup THEN
	xResistenciaSuperiorPausa02:=FALSE;
END_IF

//Liga Resistências Inferiores
xLigaResistenciaInferior:=(LigaInfPorAquecimentoReceita OR LigaInfPorAquecimentoRampa);
xLigaDeslResInferiores:= xLigaResistenciaInferior AND NOT xResistenciaInferiorPausa;
xResistenciaInferiorOn:=xLigaResistenciaInferior;

//Liga Resistências Superiores
xLigaResistenciaSuperior:= (LigaSupPorAquecimentoReceita OR LigaSupPorAquecimentoRampa);
xLigaDeslResSuperiores:= xLigaResistenciaSuperior AND NOT xResistenciaSuperiorPausa01 AND NOT xResistenciaSuperiorPausa02;
xResistenciaSuperiorOn:=xLigaResistenciaSuperior;

FOR Index:=1 TO iNumResistencias DO
	// Temperaturas Inferiores
	rTermoparInferiorLeitura[Index]:=INT_TO_REAL (TermoparLogicoInferior[Index])/10;
	rTemperaturaInferiorAtual[Index]:=(INT_TO_REAL (TermoparLogicoInferior[Index])/10);//rTemperaturaInferiorSetor[Index];
	rTermoparInferiorControle[Index]:=INT_TO_REAL (TermoparLogicoInferior[Index])/10;
	// Temperaturas Superiores
	rTermoparSuperiorLeitura[Index]:=INT_TO_REAL (TermoparLogicoSuperior[Index])/10;
	rTemperaturaSuperiorAtual[Index]:=(INT_TO_REAL (TermoparLogicoSuperior[Index])/10);//rTemperaturaSuperiorSetor[Index];
	rTermoparSuperiorControle[Index]:=INT_TO_REAL (TermoparLogicoSuperior[Index])/10;
END_FOR

// RESISTÊNCIAS INFERIORES
xLigaDesligaInfG01:= xLigaDeslResInferiores AND xAlternaSetor;
xLigaDesligaInfG02:= xLigaDeslResInferiores AND NOT xAlternaSetor;
// RESISTÊNCIAS SUPERIORES
xLigaDesligaSupG01:= xLigaDeslResSuperiores;// AND NOT xAlternaSetor;
xLigaDesligaSupG02:= xLigaDeslResSuperiores;// AND xAlternaSetor;

xHabilitaBlocosControleInferior:=xLigaDeslResInferiores;
xHabilitaBlocosControleSuperior:=xLigaDeslResSuperiores;
